// TwinCAT 3 PLC project stocker
// ProgramVersion: 3.1.4023.0
// CompilerDefines: VISU_USEWSTRING
// libraries:
//   CmpBitmapPool, * (System)
//   Tc2_MC2, * (Beckhoff Automation GmbH)
//   Tc2_Standard, * (Beckhoff Automation GmbH)
//   Tc2_System, * (Beckhoff Automation GmbH)
//   Tc2_Utilities, * (Beckhoff Automation GmbH)
//   Tc3_Module, * (Beckhoff Automation GmbH)
//   VisuDialogs, * (System)
//   VisuSymbols,3.5.10.0,System
// project tree:
//   DUTs/ENUM/ eP_alarmCode.TcDUT, eP_alarmLevel.TcDUT, eP_calculateMode.TcDUT, eP_direction.TcDUT, eP_ejevacMode.TcDUT, eP_eleMoveMode.TcDUT, eP_motionDirection.TcDUT, eP_programMode.TcDUT, eP_svMoveMode.TcDUT, eP_svType.TcDUT, eP_xyz.TcDUT
//   DUTs/REF/ ref_eje_input.TcDUT, ref_eje_io.TcDUT, ref_eje_output.TcDUT, ref_eje_param.TcDUT, ref_ele_input.TcDUT, ref_ele_io.TcDUT, ref_ele_output.TcDUT, ref_ele_param.TcDUT, ref_incjetInfo.TcDUT, ref_mc_moveAbs.TcDUT, ref_palletize.TcDUT, ref_productInfo.TcDUT, ref_sv_input.TcDUT, ref_sv_io.TcDUT, ref_sv_output.TcDUT, ref_sv_param.TcDUT, ref_teachingDetail.TcDUT, ref_teachPos.TcDUT, ref_cav.TcDUT, ref_upperLower.TcDUT, ref_XYZ.TcDUT
//   DUTs/ s_alarmList.TcDUT, s_DataSample.TcDUT, s_DataSampleCav.TcDUT, s_DataSampleCav_setQty.TcDUT, s_DataSampleGatelength.TcDUT, s_DataSamplePocketQty.TcDUT, s_gm_rotaryPos.TcDUT, s_DaraSampleSetQty.TcDUT, s_str_alarmList.TcDUT, s_timeSchedule.TcDUT, s_vels.TcDUT, s_velsXYZ.TcDUT
//   FBs/error/ fb_buzzerGenerater.TcPOU, fb_eventController.TcPOU, fb_eventListGenerator.TcPOU, fun_setAlarm.TcPOU
//   FBs/ fb_auto.TcPOU, fb_dataSampling.TcPOU, fb_debugData.TcPOU, fb_debuger.TcPOU, fb_gateLengthList.TcPOU, fb_getCav.TcPOU, fb_coordinateCal.TcPOU, fb_exchangeTraySystem.TcPOU, fb_IO.TcPOU, fb_jogController.TcPOU, fb_lsm_main.TcPOU, fb_manual.TcPOU, fb_mapping.TcPOU, fb_modeController.TcPOU, fb_motionController.TcPOU, fb_motorController.TcPOU, fb_oeprationChuck.TcPOU, fb_oeprationPush.TcPOU, fb_operationEjector.TcPOU, fb_operationElecylinder.TcPOU, fb_palletizeing.TcPOU, fb_paramInit.TcPOU, fb_productGenerator.TcPOU, fb_PTP.TcPOU, fb_recordingSystem.TcPOU, fb_sampleSchedule.TcPOU, fb_svControllers.TcPOU, fb_lensTranport.TcPOU, fb_text_control.TcPOU, fb_vacuumRetry.TcPOU, fb_eleControllers.TcPOU
//   FBs/fb_ejecter/ fb_ejector_io.TcPOU, fb_eje_controller.TcPOU, fb_eje_reset.TcPOU
//   FBs/fb_ele/ fb_ele_controller.TcPOU, fb_ele_io.TcPOU, fb_ele_reset.TcPOU
//   FBs/fb_sv/ fb_sv_controller.TcPOU, fb_sv_io.TcPOU, fb_sv_reset.TcPOU
//   FBs/gateMeasurementModule/ fb_gm_measurementModule.TcPOU, fb_gm_operationEjector.TcPOU, fb_gm_operationElecylinder.TcPOU, fb_gm_operationSV.TcPOU, fb_gm_PTP.TcPOU, fb_gm_removeLens.TcPOU, fb_gm_setting.TcPOU, fb_gm_transport.TcPOU
//   FBs/Incjet/ fb_incjetMapping.TcPOU
//   / GlobalTextList.TcGTLO, PlcTask.TcTTO, Visualization Manager.TcVMO (not stored), VISU_TASK.TcTTO
//   GVLs/ gvl_auto.TcGVL, gvl_axis.TcGVL, gvl_elecylinder.TcGVL, gvl_error.TcGVL, gvl_debug.TcGVL, gvl_gm.TcGVL, gvl_io.TcGVL, gvl_param.TcGVL, gvl_solv.TcGVL, gvl_text.TcGVL, gvl_visu.TcGVL
//   POUs/ MAIN.TcPOU
//   VISUs/Dialog/ d_gm_saveBtn.TcVIS, d_palletizeReset.TcVIS, d_preset.TcVIS, d_resetProject.TcVIS, d_sampleSchedule.TcVIS, d_saveBtn.TcVIS, d_saveProduct.TcVIS, d_saveSample.TcVIS, d_teahingDetail.TcVIS
//   VISUs/Sheet/ ImagePool.TcIPO (not stored), s_debug.TcVIS, s_gateLengthData.TcVIS, s_manual.TcVIS, s_addNewProduct.TcVIS, s_alarm.TcVIS, s_auto.TcVIS, s_gm_teaching.TcVIS, s_monitor.TcVIS, s_sample.TcVIS, s_setting.TcVIS, s_teaching1.TcVIS
// real-time tasks:
//   TASK PlcTask: cycle T#10ms, priority 20, ADS port 350
//   TASK VISU_TASK: cycle T#10ms, priority 30, ADS port 352
//   TASK VISU_TASK1: cycle T#10ms, priority 1, ADS port 351
// motion (NC):
//   TASK NC-Task 1 SAF: cycle T#2ms, priority 4, ADS port 501
//   TASK NC-Task 1 SVB: cycle T#10ms, priority 8, ADS port 511
//   AXIS lsm_axisX (id 1)
//     Velo: Maximum=5000
//     OtherSettings: AllowMotionCmdToSlave=true
//     encoder EncType=1
//       EncPara: ScaleFactorNumerator=54, ScaleFactorDenominator=10000, ReferenceSystem=1
//     drive DrvType=5
//       Analog: VeloReferenz=5200, TorqueSetpointScale=10, ScaleFactorActTorque=0.1
//       TimeComp: TaskDelayCycles=1
//     controller CtrType=1
//       CtrPara: PriorControlFactor=1
//         PosDiffControl: Enable=false
//         Observer: BandWidth=20
//   AXIS lsm_axisY (id 2)
//     Velo: Maximum=5000
//     OtherSettings: AllowMotionCmdToSlave=true
//     encoder EncType=1
//       EncPara: ScaleFactorNumerator=10, ScaleFactorDenominator=10000, ReferenceSystem=1
//     drive DrvType=5
//       Analog: VeloReferenz=5200, TorqueSetpointScale=10, ScaleFactorActTorque=0.1
//       TimeComp: TaskDelayCycles=1
//     controller CtrType=1
//       CtrPara: PriorControlFactor=1
//         PosDiffControl: Enable=false
//         Observer: BandWidth=20
//   AXIS lsm_axisZ (id 3)
//     Velo: Maximum=5000
//     OtherSettings: AllowMotionCmdToSlave=true
//     encoder EncType=1
//       EncPara: ScaleFactorNumerator=5, ScaleFactorDenominator=10000, ReferenceSystem=1
//     drive DrvType=5
//       Analog: VeloReferenz=5200, TorqueSetpointScale=10, ScaleFactorActTorque=0.1
//       TimeComp: TaskDelayCycles=1
//     controller CtrType=1
//       CtrPara: PriorControlFactor=1
//         PosDiffControl: Enable=false
//         Observer: BandWidth=20
//   AXIS gm_axisR (id 4)
//     General: UnitName=°
//     OtherSettings: AllowMotionCmdToSlave=true
//     encoder EncType=1
//       EncPara: ScaleFactorNumerator=20, ScaleFactorDenominator=10000, ReferenceSystem=1
//     drive DrvType=5
//       Analog: TorqueSetpointScale=10, ScaleFactorActTorque=0.1
//       TimeComp: TaskDelayCycles=1
//     controller CtrType=1
//       CtrPara: PriorControlFactor=1
//         Observer: BandWidth=20
// I/O:
//   DEVICE Device 1 (EtherCAT) (disabled), AmsNetId 192.168.8.53.2.1
//     Term 1 (EK1200) [EK1200-5000 EtherCAT Power supply (2A E-Bus)]
//       Term 2 (EL2088) [EL2088 8Ch. Dig. Output 24V, 0.5A, switching to negative]
//       Term 3 (EL1088) [EL1088 8Ch. Dig. Input 24V, 3ms, negative]
//       Term 4 (EK1110) [EK1110 EtherCAT extension]
//     Drive 5 (AZD4A-KED) [AZD4A-KED rev0301]
//     Box 6 (RCGW-ECT(32Byte/32Byte)) [RCGW-ECT(32Byte/32Byte)]
//     Box 7 (CU1128) [CU1128 6x EtherCAT junction]
//       Term 8 (EK1100) [EK1100 EtherCAT Coupler (2A E-Bus)]
//         Term 9 (EL2889) [EL2889 16Ch. Dig. Output 24V, 0.5A, negative]
//         Term 10 (EL2088) [EL2088 8Ch. Dig. Output 24V, 0.5A, switching to negative]
//         Term 11 (EL1889) [EL1889 16Ch. Dig. Input 24V, 3ms, negative]
//         Term 12 (EL1088) [EL1088 8Ch. Dig. Input 24V, 3ms, negative]
//         Term 17 (EL9011) [EL9011 End Terminal]
//       Box 13 (DL-EC1A) [DL-EC1A]
//       Box 14 (ECCBP88N) [ECCBP Digital 8 Inputs/8 Outputs Unit (NPN)]
//       Term 15 (CU1128-B) [CU1128 6x EtherCAT junction - Dev A]
//       Term 16 (CU1128-C) [CU1128 6x EtherCAT junction - Dev B]
// variable links:
//   stocker/stocker Instance <-> Device 1 (EtherCAT)/Box 6 (RCGW-ECT(32Byte/32Byte))
//     PlcTask Inputs/gvl_io.in_wire_ele_gateMeasurement <-> In/IN02
//     PlcTask Inputs/gvl_io.in_wire_ele_stocker <-> In/IN01
//     PlcTask Outputs/gvl_io.out_wire_ele_gateMeasurement <-> Out/OUT02
//     PlcTask Outputs/gvl_io.out_wire_ele_stocker <-> Out/OUT01
//   stocker/stocker Instance <-> Device 1 (EtherCAT)/Box 7 (CU1128)/Box 13 (DL-EC1A)
//     PlcTask Inputs/gvl_io.in_wire_gateLength <-> ID01 Current Value/ID01 Current Value (P.V.)
//     PlcTask Inputs/gvl_io.in_wire_gateMeasurementStatus <-> Status of System/Error Status
//   stocker/stocker Instance <-> Device 1 (EtherCAT)/Box 7 (CU1128)/Box 14 (ECCBP88N)
//     PlcTask Inputs/gvl_io.in_bitNumber{0..3} <-> TxPDO1/DI{4..7}  (4 links)
//     PlcTask Inputs/gvl_io.in_wire_dummySignal <-> TxPDO1/DI2
//     PlcTask Inputs/gvl_io.in_wire_gatelengthIsSuccessed <-> TxPDO1/DI1
//     PlcTask Inputs/gvl_io.in_wire_lensSetDone <-> TxPDO1/DI0
//     PlcTask Outputs/gvl_io.out_wire_requestLens <-> RxPDO1/DO0
//   stocker/stocker Instance <-> Device 1 (EtherCAT)/Box 7 (CU1128)/Term 8 (EK1100)/Term 10 (EL2088)
//     PlcTask Outputs/gvl_io.out_wire_gm_svPickUp <-> Channel 3/Output
//     PlcTask Outputs/gvl_io.out_wire_gm_svRotary <-> Channel 5/Output
//     PlcTask Outputs/gvl_io.out_wire_gm_svStamp <-> Channel 1/Output
//   stocker/stocker Instance <-> Device 1 (EtherCAT)/Box 7 (CU1128)/Term 8 (EK1100)/Term 11 (EL1889)
//     PlcTask Inputs/gvl_io.in_wire_ejectorBrk <-> Channel 9/Input
//     PlcTask Inputs/gvl_io.in_wire_ejectorVac <-> Channel 8/Input
//     PlcTask Inputs/gvl_io.in_wire_fiberSens <-> Channel 14/Input
//     PlcTask Inputs/gvl_io.in_wire_gm_ejectorBrk <-> Channel 2/Input
//     PlcTask Inputs/gvl_io.in_wire_gm_ejectorVac <-> Channel 1/Input
//     PlcTask Inputs/gvl_io.in_wire_gm_fiberSens <-> Channel 7/Input
//     PlcTask Inputs/gvl_io.in_wire_gm_svChuckClose <-> Channel 6/Input
//     PlcTask Inputs/gvl_io.in_wire_gm_svChuckOpen <-> Channel 5/Input
//     PlcTask Inputs/gvl_io.in_wire_gm_svPushClose <-> Channel 4/Input
//     PlcTask Inputs/gvl_io.in_wire_gm_svPushOpen <-> Channel 3/Input
//     PlcTask Inputs/gvl_io.in_wire_incjet_error <-> Channel 16/Input
//     PlcTask Inputs/gvl_io.in_wire_incjet_ready <-> Channel 15/Input
//     PlcTask Inputs/gvl_io.in_wire_svChuckClose <-> Channel 11/Input
//     PlcTask Inputs/gvl_io.in_wire_svChuckOpen <-> Channel 10/Input
//     PlcTask Inputs/gvl_io.in_wire_svPushClose <-> Channel 13/Input
//     PlcTask Inputs/gvl_io.in_wire_svPushOpen <-> Channel 12/Input
//   stocker/stocker Instance <-> Device 1 (EtherCAT)/Box 7 (CU1128)/Term 8 (EK1100)/Term 12 (EL1088)
//     PlcTask Inputs/gvl_io.in_wire_gm_svPickUpMoving <-> Channel 4/Input
//     PlcTask Inputs/gvl_io.in_wire_gm_svPickUpOrigin <-> Channel 3/Input
//     PlcTask Inputs/gvl_io.in_wire_gm_svRotaryMoving <-> Channel 6/Input
//     PlcTask Inputs/gvl_io.in_wire_gm_svRotaryOrigin <-> Channel 5/Input
//     PlcTask Inputs/gvl_io.in_wire_gm_svStampMoving <-> Channel 2/Input
//     PlcTask Inputs/gvl_io.in_wire_gm_svStampOrigin <-> Channel 1/Input
//   stocker/stocker Instance <-> Device 1 (EtherCAT)/Box 7 (CU1128)/Term 8 (EK1100)/Term 9 (EL2889)
//     PlcTask Outputs/gvl_io.out_wire_ejectorBrk <-> Channel 9/Output
//     PlcTask Outputs/gvl_io.out_wire_ejectorVac <-> Channel 8/Output
//     PlcTask Outputs/gvl_io.out_wire_gm_ejectorBrk <-> Channel 2/Output
//     PlcTask Outputs/gvl_io.out_wire_gm_ejectorVac <-> Channel 1/Output
//     PlcTask Outputs/gvl_io.out_wire_gm_svCPush <-> Channel 3/Output
//     PlcTask Outputs/gvl_io.out_wire_gm_svChuck <-> Channel 5/Output
//     PlcTask Outputs/gvl_io.out_wire_incjet_stampDeny <-> Channel 16/Output
//     PlcTask Outputs/gvl_io.out_wire_svCPush <-> Channel 12/Output
//     PlcTask Outputs/gvl_io.out_wire_svChuck <-> Channel 10/Output
//   stocker/stocker Instance <-> Device 1 (EtherCAT)/Term 1 (EK1200)/Term 2 (EL2088)
//     PlcTask Outputs/gvl_io.out_wire_saftyUnitReset <-> Channel 1/Output
//     PlcTask Outputs/gvl_io.out_wire_signalTowerBuzzer <-> Channel 5/Output
//     PlcTask Outputs/gvl_io.out_wire_signalTowerGreen <-> Channel 4/Output
//     PlcTask Outputs/gvl_io.out_wire_signalTowerRed <-> Channel 2/Output
//     PlcTask Outputs/gvl_io.out_wire_signalTowerYellow <-> Channel 3/Output
//   stocker/stocker Instance <-> Device 1 (EtherCAT)/Term 1 (EK1200)/Term 3 (EL1088)
//     PlcTask Inputs/gvl_io.in_wire_frontSaftyDoor <-> Channel 3/Input
//     PlcTask Inputs/gvl_io.in_wire_saftyUnitState <-> Channel 1/Input
//   stocker/stocker Instance <-> NC-Task 1 SAF/Axes/gm_axisR
//     PlcTask Inputs/gvl_axis.axisR.NcToPlc <-> Outputs/ToPlc
//     PlcTask Outputs/gvl_axis.axisR.PlcToNc <-> Inputs/FromPlc
//   stocker/stocker Instance <-> NC-Task 1 SAF/Axes/lsm_axisX
//     PlcTask Inputs/gvl_axis.axisX.NcToPlc <-> Outputs/ToPlc
//     PlcTask Outputs/gvl_axis.axisX.PlcToNc <-> Inputs/FromPlc
//   stocker/stocker Instance <-> NC-Task 1 SAF/Axes/lsm_axisY
//     PlcTask Inputs/gvl_axis.axisY.NcToPlc <-> Outputs/ToPlc
//     PlcTask Outputs/gvl_axis.axisY.PlcToNc <-> Inputs/FromPlc
//   stocker/stocker Instance <-> NC-Task 1 SAF/Axes/lsm_axisZ
//     PlcTask Inputs/gvl_axis.axisZ.NcToPlc <-> Outputs/ToPlc
//     PlcTask Outputs/gvl_axis.axisZ.PlcToNc <-> Inputs/FromPlc

CONFIGURATION stocker
    RESOURCE PLC ON TwinCAT3
        TASK PlcTask(INTERVAL := T#10ms, PRIORITY := 20);
        TASK VISU_TASK(INTERVAL := T#10ms, PRIORITY := 40);
        PROGRAM MAIN WITH PlcTask : MAIN;
        PROGRAM VisuElems_Visu_Prg WITH VISU_TASK : VisuElems.Visu_Prg;
    END_RESOURCE
END_CONFIGURATION

// ---- DUTs/ENUM/eP_alarmCode.TcDUT
{attribute 'qualified_only'}
{attribute 'strict'}
TYPE eP_alarmCode :
(
	_ := 0,
	A,
	E,
	M,
	GM,
	W
);
END_TYPE

// ---- DUTs/ENUM/eP_alarmLevel.TcDUT
{attribute 'qualified_only'}
{attribute 'strict'}
TYPE eP_alarmLevel :
(
	NONE := 0,
	INFO := 1,
	WARNING := 2,
	ERROR := 3
);
END_TYPE

// ---- DUTs/ENUM/eP_calculateMode.TcDUT
{attribute 'qualified_only'}
{attribute 'strict'}
TYPE eP_calculateMode :
(
	Affine := 0,
	Homography := 1
);
END_TYPE

// ---- DUTs/ENUM/eP_direction.TcDUT
{attribute 'qualified_only'}
{attribute 'strict'}
TYPE eP_direction :
(
	keep :=0,
	negative,
	positive
);
END_TYPE

// ---- DUTs/ENUM/eP_ejevacMode.TcDUT
{attribute 'qualified_only'}
{attribute 'strict'}
TYPE eP_ejevacMode :
(
	vacON := 1,
	vacOff := 2,
	break := 3,
	breakOff := 4,
	halt := 0
);
END_TYPE

// ---- DUTs/ENUM/eP_eleMoveMode.TcDUT
{attribute 'qualified_only'}
{attribute 'strict'}
TYPE eP_eleMoveMode :
(
	eleA := 1,
	eleB :=-1,
	stop := 0
);
END_TYPE

// ---- DUTs/ENUM/eP_motionDirection.TcDUT
{attribute 'qualified_only'}
{attribute 'strict'}
TYPE eP_motionDirection :
(
	XYZ := 1,
	ZYX := -1,
	Y_X_Z := 2,
	Z_X_Y := -2
);
END_TYPE

// ---- DUTs/ENUM/eP_programMode.TcDUT
{attribute 'qualified_only'}
{attribute 'strict'}
TYPE eP_programMode :
(
	manual := 0,
	auto,
	error
);
END_TYPE

// ---- DUTs/ENUM/eP_svMoveMode.TcDUT
{attribute 'qualified_only'}
{attribute 'strict'}
TYPE eP_svMoveMode :
(
	svA := 1,
	svB := -1,
	stop := 0
);
END_TYPE

// ---- DUTs/ENUM/eP_svType.TcDUT
{attribute 'qualified_only'}
{attribute 'strict'}
TYPE eP_svType :
(
	single,
	double
);
END_TYPE

// ---- DUTs/ENUM/eP_xyz.TcDUT
{attribute 'qualified_only'}
{attribute 'strict'}
TYPE eP_xyz :
(
	x := 0,
	y,
	z
);
END_TYPE

// ---- DUTs/REF/ref_eje_input.TcDUT
TYPE ref_eje_input :
STRUCT
	in_flg_sensVac : BOOL;
	in_flg_sensBrk : BOOL;
END_STRUCT
END_TYPE

// ---- DUTs/REF/ref_eje_io.TcDUT
TYPE ref_eje_io :
STRUCT
	param:	ref_eje_param;
	input:	ref_eje_input;
	output:	ref_eje_output;
END_STRUCT
END_TYPE

// ---- DUTs/REF/ref_eje_output.TcDUT
TYPE ref_eje_output :
STRUCT
	out_flg_ejeVac : BOOL;
	out_flg_ejeBrk : BOOL;
END_STRUCT
END_TYPE

// ---- DUTs/REF/ref_eje_param.TcDUT
TYPE ref_eje_param :
STRUCT
	var_mutex : INT;
	var_timeOut : TIME;
	var_BrkTime : TIME;
	flg_reset :BOOL;
END_STRUCT
END_TYPE

// ---- DUTs/REF/ref_ele_input.TcDUT
TYPE ref_ele_input :
STRUCT
	in_flg_sensA : BOOL;
	in_flg_sensB : BOOL;
	in_flg_sensNone : BOOL;
	in_wire_error : bool;
END_STRUCT
END_TYPE

// ---- DUTs/REF/ref_ele_io.TcDUT
TYPE ref_ele_io :
STRUCT
	param:	ref_ele_param;
	input:	ref_ele_input;
	output:	ref_ele_output;
END_STRUCT
END_TYPE

// ---- DUTs/REF/ref_ele_output.TcDUT
TYPE ref_ele_output :
STRUCT
	out_flg_eleA : BOOL;
	out_flg_eleB : BOOL;
	out_flg_reset : BOOL;
END_STRUCT
END_TYPE

// ---- DUTs/REF/ref_ele_param.TcDUT
TYPE ref_ele_param :
STRUCT
	var_mutex : INT;
	var_timeOut : TIME;
	flg_reset :BOOL;
END_STRUCT
END_TYPE

// ---- DUTs/REF/ref_incjetInfo.TcDUT
TYPE ref_incjetInfo :
STRUCT
	var_msgNo : INT;
	flg_denyStamp : BOOL;
	flg_numberingReset : BOOL;
	flg_numberingCount : BOOL;
	flg_numberingStop : BOOL;
	flg_warningReset : BOOL;
	flg_stampReady : BOOL;
	flg_incLow : BOOL;
	flg_incOut : BOOL;
	flg_error : BOOL;
	flg_busy : BOOL;
	flg_stampRun : BOOL;
	flg_heatUpDone : BOOL;
	flg_systemRun : BOOL;
	flg_stampsDone : BOOL;
	flg_numberingCountDone : BOOL;
	flg_fluxLow : BOOL;
	flg_incFluxLow : BOOL;
	flg_headCoverIsOpen : BOOL;
	flg_stampDone : BOOL;
END_STRUCT
END_TYPE

// ---- DUTs/REF/ref_mc_moveAbs.TcDUT
TYPE ref_mc_moveAbs :
STRUCT
	Execute      : BOOL;
    Position     : LREAL; 
    Velocity     : LREAL; 
    Acceleration : LREAL; 
    Deceleration : LREAL; 
    Jerk         : LREAL;
    BufferMode   : MC_BufferMode;
    Options      : ST_MoveOptions;
	Done           : BOOL;
    Busy           : BOOL;
    Active         : BOOL;
    CommandAborted : BOOL;
    Error          : BOOL;
    ErrorID        : UDINT;
END_STRUCT
END_TYPE

// ---- DUTs/REF/ref_palletize.TcDUT
TYPE ref_palletize :
STRUCT
	Pos : ARRAY[1..4] OF ref_xyz ;
	teachingDetail : ref_teachingDetail;
	teachingDetailVels : s_velsXYZ;
END_STRUCT
END_TYPE

// ---- DUTs/REF/ref_productInfo.TcDUT
TYPE ref_productInfo :
STRUCT
	num : INT;
	name : STRING;
	cavQty : INT;
	bottomPocketQty : INT;
	vertivalPocketQty : INT ;
	pocketSumQty : INT;
	startCav : INT;
	gateLength_min : INT;
	gateLength_max : INT;
	teachPos : ref_teachPos;
	autoVels : s_velsXYZ;
	manaulVels : s_velsXYZ;
	incjetMsgNo : INT;
	flg_mode_stocker: BOOL;
	flg_mode_measurement: BOOL;
END_STRUCT
END_TYPE

// ---- DUTs/REF/ref_sv_input.TcDUT
TYPE ref_sv_input :
STRUCT
	in_flg_sensA:	BOOL;
	in_flg_sensB:	BOOL;
END_STRUCT
END_TYPE

// ---- DUTs/REF/ref_sv_io.TcDUT
TYPE ref_sv_io :
STRUCT
	param: ref_sv_param;
	in: ref_sv_input;
	out:ref_sv_output;
END_STRUCT
END_TYPE

// ---- DUTs/REF/ref_sv_output.TcDUT
TYPE ref_sv_output :
STRUCT
	out_flg_svA:	BOOL;
	out_flg_svB:	BOOL;
END_STRUCT
END_TYPE

// ---- DUTs/REF/ref_sv_param.TcDUT
TYPE ref_sv_param :
STRUCT
	var_svType:ep_svType;
	var_mutex : INT;
	var_timeOut : TIME;
	flg_reset :BOOL;
END_STRUCT
END_TYPE

// ---- DUTs/REF/ref_teachingDetail.TcDUT
TYPE ref_teachingDetail :
STRUCT
	passingPos : ref_XYZ;
	settingPos : ref_XYZ;
END_STRUCT
END_TYPE

// ---- DUTs/REF/ref_teachPos.TcDUT
TYPE ref_teachPos :
STRUCT
	palletize : ref_upperLower;
	initial : ref_xyz;
	pickUp : ref_xyz;
	remove :ref_xyz;
	sample  : ARRAY[1..8] OF ref_xyz;
	gm_rotary	: s_gm_rotaryPos;
END_STRUCT
END_TYPE

// ---- DUTs/REF/ref_cav.TcDUT
TYPE ref_cav :
STRUCT
	cav : ARRAY [1..8] OF  ref_palletize;
END_STRUCT
END_TYPE

// ---- DUTs/REF/ref_upperLower.TcDUT
TYPE ref_upperLower :
STRUCT
	upperLower : ARRAY[1..2] OF ref_cav ;
END_STRUCT
END_TYPE

// ---- DUTs/REF/ref_XYZ.TcDUT
TYPE ref_XYZ :
STRUCT
	x : LREAL ;
	y : LREAL ;
	z : LREAL ;
END_STRUCT
END_TYPE

// ---- DUTs/s_alarmList.TcDUT
TYPE s_alarmList :
STRUCT
	var_alarmLevel : eP_alarmLevel;
	var_alarmName : WSTRING;
	var_alarmMassge : WSTRING;
	var_alarmTime : DT;
	var_alarmCode1 : eP_alarmCode;
	var_alarmCode2 : UDINT;
	
END_STRUCT
END_TYPE

// ---- DUTs/s_DataSample.TcDUT
TYPE s_DataSample :
STRUCT
	DataSet :  ARRAY[0..500] OF s_DataSampleCav;
	SetQty	:  s_DataSampleCav_setQty;
END_STRUCT
END_TYPE

// ---- DUTs/s_DataSampleCav.TcDUT
TYPE s_DataSampleCav :
STRUCT
	cav : ARRAY[0..8] OF s_DataSamplePocketQty;
END_STRUCT
END_TYPE

// ---- DUTs/s_DataSampleCav_setQty.TcDUT
TYPE s_DataSampleCav_setQty :
STRUCT
	cav : ARRAY[0..8] OF  s_DaraSampleSetQty;
END_STRUCT
END_TYPE

// ---- DUTs/s_DataSampleGatelength.TcDUT
TYPE s_DataSampleGatelength :
STRUCT
	gateLength	: LREAL;
	setDate		: STRING;
END_STRUCT
END_TYPE

// ---- DUTs/s_DataSamplePocketQty.TcDUT
TYPE s_DataSamplePocketQty :
STRUCT
	pocketNo : ARRAY[0..100] OF s_DataSampleGatelength;
END_STRUCT
END_TYPE

// ---- DUTs/s_gm_rotaryPos.TcDUT
TYPE s_gm_rotaryPos :
STRUCT
	origin	: LREAL;
	pickUp	: LREAL;
	set		: LREAL;
	remove  : LREAL;
END_STRUCT
END_TYPE

// ---- DUTs/s_DaraSampleSetQty.TcDUT
TYPE s_DaraSampleSetQty :
STRUCT
	nonDefectiveQty : INT;
	defectiveQty	:INT;
END_STRUCT
END_TYPE

// ---- DUTs/s_str_alarmList.TcDUT
TYPE s_str_alarmList :
STRUCT
	var_alarmLevel : STRING;
	var_alarmName : WSTRING;
	var_alarmMassge : WSTRING;
	var_alarmTime : STRING;
	var_alarmCode1 : eP_alarmCode;
	var_alarmCode2 : STRING;
	
END_STRUCT
END_TYPE

// ---- DUTs/s_timeSchedule.TcDUT
TYPE s_timeSchedule :
STRUCT
	hour : WORD;
	minute: WORD;
END_STRUCT
END_TYPE

// ---- DUTs/s_vels.TcDUT
TYPE s_vels :
STRUCT
	vel : LREAL := 20;
	acc : LREAL := 20;
	dcc : LREAL := 20;
END_STRUCT
END_TYPE

// ---- DUTs/s_velsXYZ.TcDUT
TYPE s_velsXYZ :
STRUCT
	x : s_vels;
	y : s_vels;
	z : s_vels;
END_STRUCT
END_TYPE

// ---- GVLs/gvl_auto.TcGVL
{attribute 'qualified_only'}
VAR_GLOBAL
	gateLengthIsPassed		: BOOL;
	requirementToPickUpLens	: BOOL;
	pickUpLnesDone			: BOOL;
	chuckopenDone			: BOOL;
	lensVacuumDone			: BOOL;
	cavNo					: INT;
	buf_cavNo				: INT ;
	autoModeStop			: BOOL;
	autoModeStoped			: BOOL;
	motorPowerOn			: BOOL;
	flg_trayChangeDone		: BOOL;
	gm_rotaryPowerOn		: BOOL;
	flg_gateData_Tx			: BOOL;
	flg_gm_measurementClosed: BOOL;
	flg_gm_transportClosed	: BOOL;
	flg_transportClosed		: BOOL;
	flg_VacuumRetry			: BOOL;
	flg_gm_VacuumRetry		: BOOL;
	flg_DataSample_nonDefective: BOOL;
	flg_DataSample_defective: BOOL;
	flg_DataSamle_sample: BOOL;
	buf_gateLength: LREAL;
	flg_dataSampling_run: BOOL;
	var_DataSet				: s_DataSample; //lateset data is var_DataSet[0], oldest is var_DataSet[500], cav[0] and pocketNo[0] are unused
	flg_gm_eleIsDown: BOOL;
	flg_axisIsPcikingUp: BOOL;
	flg_buf_gateLengthIsPassed: BOOL;
	flg_gateLength: BOOL;
	flg_sampling: BOOL;
END_VAR
VAR_GLOBAL PERSISTENT
	pocketNo				: ARRAY[0..8] OF INT;
	var_defectiveLens		: ARRAY[0..8] OF INT;
	
	flg_pocketCountCheck_cav: int;
	flg_pocketCountCheck: BOOL;
END_VAR

// ---- GVLs/gvl_axis.TcGVL
{attribute 'qualified_only'}
VAR_GLOBAL
	axisX : AXIS_REF;
	axisY : AXIS_REF;
	axisZ : AXIS_REF;
	axisR : AXIS_REF;
	
	fbi_mc_powerX :MC_Power;
	fbi_mc_powerY :MC_Power;
	fbi_mc_powerZ :MC_Power;
	fbi_mc_powerR :MC_Power;
	
	fbi_mc_absX : MC_MoveAbsolute;
	fbi_mc_absY : MC_MoveAbsolute;
	fbi_mc_absZ : MC_MoveAbsolute;
	fbi_mc_absR : MC_MoveAbsolute;
	
	ref_x : ref_mc_moveAbs;
	ref_y : ref_mc_moveAbs;
	ref_z : ref_mc_moveAbs;
	ref_r : ref_mc_moveAbs;
	
	fbi_mc_jogX : MC_Jog;
	fbi_mc_jogY : MC_Jog;
	fbi_mc_jogZ : MC_Jog;
	fbi_mc_jogR : MC_Jog;
	
	fbi_motionControler: fb_motionController;
	
	flg_motorReady: BOOL;
END_VAR

// ---- GVLs/gvl_elecylinder.TcGVL
{attribute 'qualified_only'}
VAR_GLOBAL
	
	fbi_axisTransport 		: fb_ele_controller;
	fbi_axisSample 			: fb_ele_controller;
	fbi_axisTrayChange 		: fb_ele_controller;
	fbi_axisRotary 			: fb_ele_controller;
	fbi_gm_axisTransport 	: fb_ele_controller;
	fbi_gm_axisPickUp 		: fb_ele_controller;
	

	ref_axis_transport 		: ref_ele_io;
	ref_axis_sample		 	: ref_ele_io;
	ref_axis_trayChange 	: ref_ele_io;
	ref_axis_rotary 		: ref_ele_io;
	ref_gm_axisTransport 	: ref_ele_io;
	ref_gm_axisPickUp 		: ref_ele_io;
END_VAR

// ---- GVLs/gvl_error.TcGVL
{attribute 'qualified_only'}
VAR_GLOBAL
	var_ary_alarmlistActive 	: ARRAY[1..10] OF s_str_alarmList;
	flg_error					: BOOL;
	flg_warning					: BOOL;
	flg_info					: BOOL;
	flg_reset					: BOOL;
	flg_alramBusy				: BOOL;
	
	flg_fiberSens 				: BOOL;
	flg_vacuum					: BOOL;
	flg_axisXTorqueOver			: BOOL;
	flg_axisYTorqueOver			: BOOL;
	flg_axisZTorqueOver			: BOOL;
	flg_axisRTorqueOver			: BOOL;
	
	flg_resetEventFlg			: BOOL;
	flg_eventDisplayRest		: BOOL;
	flg_ararmLevelRest			: BOOL;
	flg_gm_fiberSens			: BOOL;
	flg_trayChangeError			: BOOL;
	flg_incjet					: BOOL;
	
	flg_sample_windown_warning  : BOOL;
	flg_sample_windown_error	: BOOL;
END_VAR
VAR_GLOBAL PERSISTENT
	var_ary_alarmlistLog 		: ARRAY[1..50] OF s_alarmList;
END_VAR

// ---- GVLs/gvl_debug.TcGVL
{attribute 'qualified_only'}
VAR_GLOBAL
	gateLengthISSuccessed	: BOOL;
	dummySignal				: BOOL;
	lensSetDone				: BOOL;
	flg_debug_run			: BOOL;
	var_cav					: INT;
	out_busy			    : BOOL;
	out_lensSetDone			: BOOL;
	out_fiberSens			: BOOL;
	cavConecctSkip			: BOOL;
	flg_passingMeasurement	: BOOL;
	flg_stampReady: BOOL;
	flg_stampDone: BOOL;
	flg_check_quality: BOOL;
	flg_to_measurement : BOOL;
	flg_to_stocker : BOOL;
	flg_to_demand: BOOL;
	flg_to_acquired: BOOL;
	
END_VAR

// ---- GVLs/gvl_gm.TcGVL
{attribute 'qualified_only'}
VAR_GLOBAL
	
	flg_lensSetDoneFromGM		: BOOL;
	flg_lensPickUpDone			: BOOL;
	flg_requestPickup			: BOOL;
	flg_lensRequest				: BOOL;
	
	var_buf_measurementCav		: INT;
	var_buf_tranportCav			: INT;
	flg_gateLengthIsPassed: BOOL;
	flg_buf_gateLengthIsPassed: BOOL;
END_VAR
VAR_GLOBAL PERSISTENT
	var_buf_manualVel			: LREAL;
	var_buf_autoVel				: LREAL;
	var_buf_autoAcc				: LREAL;
	var_buf_autoDec				: LREAL;
	var_rotaryPos 				: s_gm_rotaryPos;
	var_incjetInfo				:ref_incjetInfo;
END_VAR

// ---- GVLs/gvl_io.TcGVL
{attribute 'qualified_only'}
VAR_GLOBAL
	in_wire_saftyCircuitState				AT %I* : BOOL;
	in_wire_saftyUnitState					AT %I* : BOOL;
	in_wire_frontSaftyDoor					AT %I* : BOOL;
	in_wire_btnGreen						AT %I* : BOOL;
	in_wire_btnRed							AT %I* : BOOL;
	in_bitNumber0							AT %I* : BOOL;
	in_bitNumber1							AT %I* : BOOL;
	in_bitNumber2							AT %I* : BOOL;
	in_bitNumber3							AT %I* : BOOL;
	in_wire_gateLengthIsFailed				AT %I* : BOOL;
	in_wire_lensSetDone						AT %I* : BOOL;
	in_wire_gatelengthIsSuccessed			AT %I* : BOOL;
	in_wire_dummySignal						AT %I* : BOOL;
	in_wire_fiberSens						AT %I* : BOOL;
	in_wire_gm_fiberSens					AT %I* : BOOL;
	//solv
	in_wire_ejectorVac						AT %I* : BOOL;
	in_wire_ejectorBrk						AT %I* : BOOL;
	in_wire_svChuckClose					AT %I* : BOOL;
	in_wire_svChuckOpen						AT %I* : BOOL;
	in_wire_svPushClose						AT %I* : BOOL;
	in_wire_svPushOpen						AT %I* : BOOL;
	in_wire_gm_ejectorVac					AT %I* : BOOL;
	in_wire_gm_ejectorBrk					AT %I* : BOOL;
	in_wire_gm_svChuckClose					AT %I* : BOOL;
	in_wire_gm_svChuckOpen					AT %I* : BOOL;
	in_wire_gm_svPushClose					AT %I* : BOOL;
	in_wire_gm_svPushOpen					AT %I* : BOOL;
	in_wire_gm_svRotaryOrigin				AT %I* : BOOL;
	in_wire_gm_svRotaryMoving				AT %I* : BOOL;
	in_wire_gm_svPickUpOrigin				AT %I* : BOOL;
	in_wire_gm_svPickUpMoving				AT %I* : BOOL;
	in_wire_gm_svStampOrigin				AT %I* : BOOL;
	in_wire_gm_svStampMoving				AT %I* : BOOL;
	//elecylinder
	in_wire_ele_stocker						AT %I* : UINT;
	in_wire_ele_gateMeasurement				AT %I* : UINT;
	
	in_wire_incjet_ready					AT %I* : BOOL;
	in_wire_incjet_run  					AT %I* : BOOL;
	in_wire_incjet_error					AT %I* : BOOL;
	
	in_flg_eleTransportOrigin						: BOOL;
	in_flg_eleTransportMoving						: BOOL;
	in_flg_eleTransportError						: BOOL;
	in_flg_eleSampleOrigin							: BOOL;
	in_flg_eleSampleMoving							: BOOL;
	in_flg_eleSampleError							: BOOL;
	in_flg_eleTrayChangeOrigin						: BOOL;
	in_flg_eleTrayChangeMoving						: BOOL;
	in_flg_eleTrayChangeError						: BOOL;
	in_flg_eleRotaryOrigin							: BOOL;
	in_flg_eleRotaryMoving							: BOOL;
	in_flg_eleRotaryError							: BOOL;
	in_flg_gm_elePickupOrigin						: BOOL;
	in_flg_gm_elePickupMoving						: BOOL;
	in_flg_gm_elePickupError						: BOOL;
	in_flg_gm_eleTransportOrigin					: BOOL;
	in_flg_gm_eleTransportMoving					: BOOL;
	in_flg_gm_eleTransPortError						: BOOL;
	
	
	
	in_wire_gateLength						AT %I* : DINT;
	in_wire_gateMeasurementStatus			AT %I* : BOOL;
	in_wire_gateMeasurementErrCode			AT %I* : UINT;
	out_wire_gateMeasurementReset			AT %Q* : DINT;
	out_wire_gateMeasurementPreset			AT %Q* : DINT;
	
	out_wire_saftyUnitReset					AT %Q* : BOOL;
	out_wire_signalTowerRed 				AT %Q* : BOOL;
	out_wire_signalTowerGreen 				AT %Q* : BOOL;
	out_wire_signalTowerYellow				AT %Q* : BOOL;
	out_wire_signalTowerBuzzer 				AT %Q* : BOOL;
	
	out_wire_requestLens					AT %Q* : BOOL;
	//solv
	out_wire_ejectorVac						AT %Q* : BOOL;
	out_wire_ejectorBrk						AT %Q* : BOOL;
	out_wire_svChuck						AT %Q* : BOOL;
	out_wire_svCPush						AT %Q* : BOOL;
	out_wire_gm_ejectorVac					AT %Q* : BOOL;
	out_wire_gm_ejectorBrk					AT %Q* : BOOL;
	out_wire_gm_svChuck						AT %Q* : BOOL;
	out_wire_gm_svCPush						AT %Q* : BOOL;
	out_wire_gm_svRotary					AT %Q* : BOOL;
	out_wire_gm_svPickUp					AT %Q* : BOOL;
	out_wire_gm_svStamp						AT %Q* : BOOL;

	//elecylinder
	out_wire_ele_stocker					AT %Q* : UINT;
	out_wire_ele_gateMeasurement			AT %Q* : UINT;
	
	out_wire_incjet_stampDeny				AT %Q* : BOOL;
	
	out_flg_eleTransportOrigin						: BOOL;
	out_flg_eleTransportMoving						: BOOL;
	out_flg_eleTransportReset						: BOOL;
	out_flg_eleSampleOrigin							: BOOL;
	out_flg_eleSampleMoving							: BOOL;
	out_flg_eleSampleReset							: BOOL;
	out_flg_eleTrayChangeOrigin						: BOOL;
	out_flg_eleTrayChangeMoving						: BOOL;
	out_flg_eleTrayChangeReset						: BOOL;
	out_flg_eleRotaryOrigin							: BOOL;
	out_flg_eleRotaryMoving							: BOOL;
	out_flg_eleRotaryReset							: BOOL;
	out_flg_gm_elePickupOrigin						: BOOL;
	out_flg_gm_elePickupMoving						: BOOL;
	out_flg_gm_elePickupReset						: BOOL;
	out_flg_gm_eleTransportOrigin					: BOOL;
	out_flg_gm_eleTransportMoving					: BOOL;
	out_flg_gm_eleTransPortReset					: BOOL;
	flg_bitNumber0									: BOOL;
	flg_bitNumber1									: BOOL;
	flg_bitNumber2									: BOOL;
	flg_bitNumber3									: BOOL;
	flg_dummySiganl									: BOOL;
	flg_gateLengthIsSuccessed						: BOOL;
	flg_lensSetDone									: BOOL;
	flg_fiberSens									: BOOL;
	flg_btnGreen									: BOOL;
	flg_btnRed										: BOOL;
	flg_frontSaftyDoor								: BOOL;
	var_gateLength									: DINT;
	flg_gatemeasurementStatus						: BOOL;
	var_gateMeasurementErrCode						: UDINT;
	var_gateMeasurementReset						: DINT;
	var_gateMeasurementPreset						: DINT;
	flg_gm_fiberSens								: BOOL;
	flg_saftyUnitState								: BOOL;
	flg_saftyUnitReset								: BOOL;
	flg_requestLens									: BOOL;
	flg_signalTowerBuzzer							: BOOL;
	flg_signalTowerGreen							: BOOL;
	flg_signalTowerRed								: BOOL;
	flg_signalTowerYellow							: BOOL;

END_VAR

// ---- GVLs/gvl_param.TcGVL
{attribute 'qualified_only'}
VAR_GLOBAL
	var_currentMode 		: eP_programMode;
	var_currentTrayPos 		: INT;
END_VAR
VAR_GLOBAL PERSISTENT
	var_productInfo 		: ARRAY [0..10] OF ref_productInfo;
	var_currentProductID 	: INT := 0;
	var_b					: INT;
END_VAR

// ---- GVLs/gvl_solv.TcGVL
{attribute 'qualified_only'}
VAR_GLOBAL	
	fbi_ejector 	: fb_eje_controller;
	fbi_chuck 		: fb_sv_controller;
	fbi_push 		: fb_sv_controller;
	fbi_gm_ejector 	: fb_eje_controller;
	fbi_gm_chuck 	: fb_sv_controller;
	fbi_gm_push 	: fb_sv_controller;
	fbi_gm_rotary 	: fb_sv_controller;
	fbi_gm_pickup 	: fb_sv_controller;
	fbi_gm_stamp 	: fb_sv_controller;

	ref_ejector 	: ref_eje_io;
	ref_chuck 		: ref_sv_io;
	ref_push 		: ref_sv_io;
	ref_gm_ejctor 	: ref_eje_io;
	ref_gm_chuck 	: ref_sv_io;
	ref_gm_push 	: ref_sv_io;
	ref_gm_rotary 	: ref_sv_io;
	ref_gm_pickUp 	: ref_sv_io;
	ref_gm_stamp 	: ref_sv_io;
END_VAR

// ---- GVLs/gvl_text.TcGVL
{attribute 'qualified_only'}
VAR_GLOBAL
	var_auto_runing: WSTRING(255);
	var_stopping: WSTRING(255);
	var_trayChangeDone: WSTRING(255);
END_VAR

// ---- GVLs/gvl_visu.TcGVL
{attribute 'qualified_only'}
VAR_GLOBAL
	flg_powerOn	: BOOL;
	var_jofAxis : eP_xyz;
	flg_btn_moveDirct : eP_direction;
	flg_btn_PosInit: BOOL;
	flg_btn_PosPickUP: BOOL;
	flg_btn_PosRemove: BOOL;
	flg_btn_PosSample: BOOL;
	flg_btn_PosPocket: BOOL;
	var_in_sampleCavNo: INT := 1;
	var_in_cavNo: INT := 1;
	var_in_pocketNo: INT := 1;
	var_in_samplePos: ref_xyz;
	var_in_initialPos: ref_xyz;
	var_in_removePos: ref_xyz;
	var_in_pickUpPos: ref_xyz;
	var_in_productGenerate: ref_productInfo;
	flg_btn_saveProductInfo: BOOL;
	flg_btn_eleTransportPostive: BOOL;
	flg_btn_eleTransportNegative: BOOL;
	flg_btn_eleSamplePositive: BOOL;
	flg_btn_eleSampleNegative: BOOL;
	flg_btn_eleTrayChangePositive: BOOL;
	flg_btn_eleTrayChangeNegative: BOOL;
	flg_btn_eleRotaryPositive: BOOL;
	flg_btn_eleRotaryNegative: BOOL;
	flg_btn_gm_elePickUpPositive: BOOL;
	flg_btn_gm_elePickUpNegative: BOOL;
	flg_btn_gm_eleTransportPositive: BOOL;
	flg_btn_gm_eleTransportNegative: BOOL;
	flg_btn_svChuckOpen: BOOL;
	flg_btn_svChuckClose: BOOL;
	flg_btn_svPushClose: BOOL;
	flg_btn_svPushOpen: BOOL;
	flg_btn_gm_svChuckOpen: BOOL;
	flg_btn_gm_svChuckClose: BOOL;
	flg_btn_gm_svPushClose: BOOL;
	flg_btn_gm_svPushOpen: BOOL;
	flg_btn_gm_svRotaryOrigin: BOOL;
	flg_btn_gm_svRotaryMoving: BOOL;
	flg_btn_gm_svPickUpOrigin: BOOL;
	flg_btn_gm_svPickUpMoving: BOOL;
	flg_btn_gm_svStampOrigin: BOOL;
	flg_btn_gm_svStampMoving: BOOL;
	flg_btn_vacuumOn: BOOL;
	flg_btn_vacuumOff: BOOL;
	flg_btn_breakOn: BOOL;
	flg_btn_gm_vacuumOn: BOOL;
	flg_btn_gm_vacuumOff: BOOL;
	flg_btn_gm_breakOn: BOOL;
	flg_btn_savePalletize: BOOL;
	flg_btn_saveSample: BOOL;
	flg_btn_sample: BOOL;
	flg_btn_autoModeStop: BOOL;
	flg_btn_gm_motorPower: BOOL;
	flg_btn_vacSensOn: BOOL;
	flg_btn_vacRobotOn: BOOL;
	flg_btn_lensSetDone: BOOL;
	var_DT: DT;
	flg_btn_clrDefectiveQty: BOOL;
	flg_btn_autoModeStart: BOOL;
	flg_btn_trayChangeDone: BOOL;
	var_msg: WSTRING;
	var_dev_passingPosY: LREAL;
	var_dev_passingPosX: LREAL;
	var_dev_passingPosZ: LREAL;
	var_dev_settingPosX: LREAL;
	var_dev_settingPosY: LREAL;
	var_dev_settingPosZ: LREAL;
	var_in_teachingDetail: ref_teachingDetail;
	var_gm_rotaryInch: LREAL;
	flg_btn_rotaryRigt: BOOL;
	flg_btn_rotaryLeft: BOOL;
	var_radio_rotaryJogMode: INT;
	flg_btn_clrPockertQty: BOOL;
	var_rotaryPos: s_gm_rotaryPos;
	flg_btn_rotaryPos: BOOL;
	flg_btn_gm_moveOrigin: BOOL;
	flg_btn_gm_movePickUp: BOOL;
	flg_btn_gm_moveSet: BOOL;
	flg_btn_gm_moveRemove: BOOL;
	var_in_teachingDetailVels: s_velsXYZ;
	var_currentTableMsg : WSTRING;
	var_curenntGateData: LREAL;
	flg_btn_projectReset: BOOL;
	flg_btn_invalidBuzzer: BOOL;
	flg_btn_gateMeasurementPreset: BOOL;
	var_projectResetLastTime: LREAL;
	flg_btn_clrGateData: BOOL;
	flg_btn_buzzer_silent: BOOL;
	flg_btn_All_PosPocket: BOOL;
	flg_All_PosPorket_Move: BOOL;
END_VAR
VAR_GLOBAL PERSISTENT
	var_in_palletizePos: ref_palletize;
	var_radio_jogMode: INT;
	var_in_inch: LREAL:=0.2;
	var_in_currentProduct : ARRAY[0..10] OF STRING;
	flg_btn_usingMeasurementSystem : BOOL;
	flg_btn_gateMeasurementIsNone: BOOL;
	var_dev_palletizingMode: BOOL;
	var_gm_manualRotaryVel: LREAL;
	var_gm_autoRotaryVel: LREAL;
	var_gm_autoRotaryAcc: LREAL;
	var_gm_autoRotaryDec: LREAL;
	var_gateLengthList: ARRAY[0..49] OF REAL;
	var_gateLengthListCav: ARRAY[1..8] OF ARRAY[0..49] OF REAL;
	flg_btn_rotaryReversal: BOOL;
	flg_btn_RotaryIsNotUse: BOOL;
	flg_missingParts: BOOL;
	flg_usingTimeStamp : BOOL;
	var_enableSchedule: ARRAY[0..6] OF BOOL;
	var_scheduleTimeH : ARRAY[0..6] OF WORD;
	var_scheduleTimeM : ARRAY[0..6] OF WORD;
END_VAR

// ---- POUs/MAIN.TcPOU
PROGRAM MAIN
VAR
	fbi_lsm_main: fb_lsm_main;
	fbi_text_control_run: fb_text_control;
END_VAR

fbi_lsm_main();
fbi_text_control_run();

END_PROGRAM

// ---- FBs/fb_lsm_main.TcPOU
FUNCTION_BLOCK fb_lsm_main
VAR_INPUT
END_VAR
VAR_OUTPUT
END_VAR
VAR
	fbi_mapping			:fb_mapping;
	fbi_IO				:fb_IO;
	fbi_modeController	:fb_modeController;
	fbi_motorController	:fb_motorController;
	fbi_eventController	:fb_eventController;
	fbi_eleControllers	:fb_eleControllers;
	fbi_svControllers	:fb_svControllers;
	fbi_recordingSystem :fb_recordingSystem;
	fbi_GetLocalAmsNetId: FB_GetLocalAmsNetId;
	fbi_LocalSystemTime: FB_LocalSystemTime;
	fbi_resetDelay: TON;
	fb_Shutdown: NT_Shutdown;
	fb_Reboot: NT_Reboot;
	ShutdownStart: BOOL;
	RebootStart: BOOL;
	fbi_WritePersistentData: FB_WritePersistentData;
	var_lastTIme: LREAL;
	gvl_error_reset: BOOL;
	fbi_productGenerater: fb_productGenerator;
	fbi_sampleSchedule: fb_sampleSchedule;
	test_flg: BOOL;
END_VAR

THIS^.fbi_mapping();
THIS^.fbi_IO();
THIS^.fbi_modeController();
THIS^.fbi_eleControllers();
THIS^.fbi_svControllers();
THIS^.fbi_recordingSystem();
THIS^.fbi_productGenerater();
THIS^.fbi_motorController();
THIS^.fbi_eventController(in_flg_run:=TRUE , out_flg_run=> );
THIS^.fbi_modeController.p_init := fbi_resetDelay.Q ;
gvl_axis.fbi_motionControler.p_Init := gvl_param.var_currentMode = eP_programMode.error;
fbi_resetDelay(IN:= gvl_visu.flg_btn_projectReset , PT:=T#5S , Q=> , ET=>  );
gvl_visu.var_projectResetLastTime :=(LREAL#5000 - TIME_TO_LREAL(fbi_resetDelay.ET))/1000;
gvl_axis.fbi_motionControler(
	in_flg_run:= TRUE, 
	out_flg_run=> , 
	var_ref_X:= gvl_axis.ref_x, 
	var_ref_Y:= gvl_axis.ref_y, 
	var_ref_Z:= gvl_axis.ref_z, 
	in_flg_start:= gvl_axis.fbi_motionControler.in_flg_start, 
	in_var_targetPosX:= , 
	in_var_targetPosY:= , 
	in_var_targetPosZ:= , 
	in_var_direction:= , 
	out_flg_busy=> , 
	out_flg_Done=> , 
	out_flg_moveXYDone=> );
fbi_sampleSchedule(in_var_enableSchedule:= gvl_visu.var_enableSchedule ,
	in_var_scheduleTimeH:= gvl_visu.var_scheduleTimeH ,
	in_var_scheduleTimeM:= gvl_visu.var_scheduleTimeM ,
	out_flg_sampletriger=> );
	IF fbi_sampleSchedule.out_flg_sampletriger AND gvl_param.var_currentMode = eP_programMode.auto THEN
		gvl_visu.flg_btn_sample := TRUE;
	END_IF
fbi_GetLocalAmsNetId(
	bExecute:=TRUE , 
	tTimeOut:= ,
	bBusy=> , 
	bError=> , 
	nErrId=> , 
	AddrString=> , 
	AddrBytes=> );
fbi_LocalSystemTime(
	sNetID:=fbi_GetLocalAmsNetId.AddrString , 
	bEnable:= TRUE, 
	dwCycle:= , 
	dwOpt:= , 
	tTimeout:= , 
	bValid=> , 
	systemTime=> , 
	tzID=> );
fb_Shutdown(
	NETID:= fbi_GetLocalAmsNetId.AddrString, 
	DELAY:= 3, 
	START:= ShutdownStart, 
	TMOUT:= T#6S, 
	BUSY=> , 
	ERR=> , 
	ERRID=> );

fb_Reboot(
	NETID:= fbi_GetLocalAmsNetId.AddrString, 
	DELAY:= 3, 
	START:= RebootStart, 
	TMOUT:= T#6S, 
	BUSY=> , 
	ERR=> , 
	ERRID=> );
fbi_WritePersistentData(
	NETID:= fbi_GetLocalAmsNetId.AddrString, 
	PORT:= 851, 
	START:= gvl_axis.fbi_motionControler.out_flg_Done, 
	TMOUT:= , 
	MODE:= , 
	BUSY=> , 
	ERR=> , 
	ERRID=> );
gvl_visu.var_DT := SYSTEMTIME_TO_DT(fbi_LocalSystemTime.systemTime);
gvl_visu.var_curenntGateData := DINT_TO_LREAL(gvl_io.var_gateLength)/10000;

END_FUNCTION_BLOCK

// ---- FBs/fb_mapping.TcPOU
FUNCTION_BLOCK fb_mapping
VAR_INPUT
END_VAR
VAR_OUTPUT
END_VAR
VAR
	fbi_ejector_io: ARRAY[1..3] OF fb_ejector_io;
	fbi_sv_io: ARRAY[1..8] OF  fb_sv_io;
	fbi_ele_io: ARRAY[1..6] OF  fb_ele_io;
END_VAR

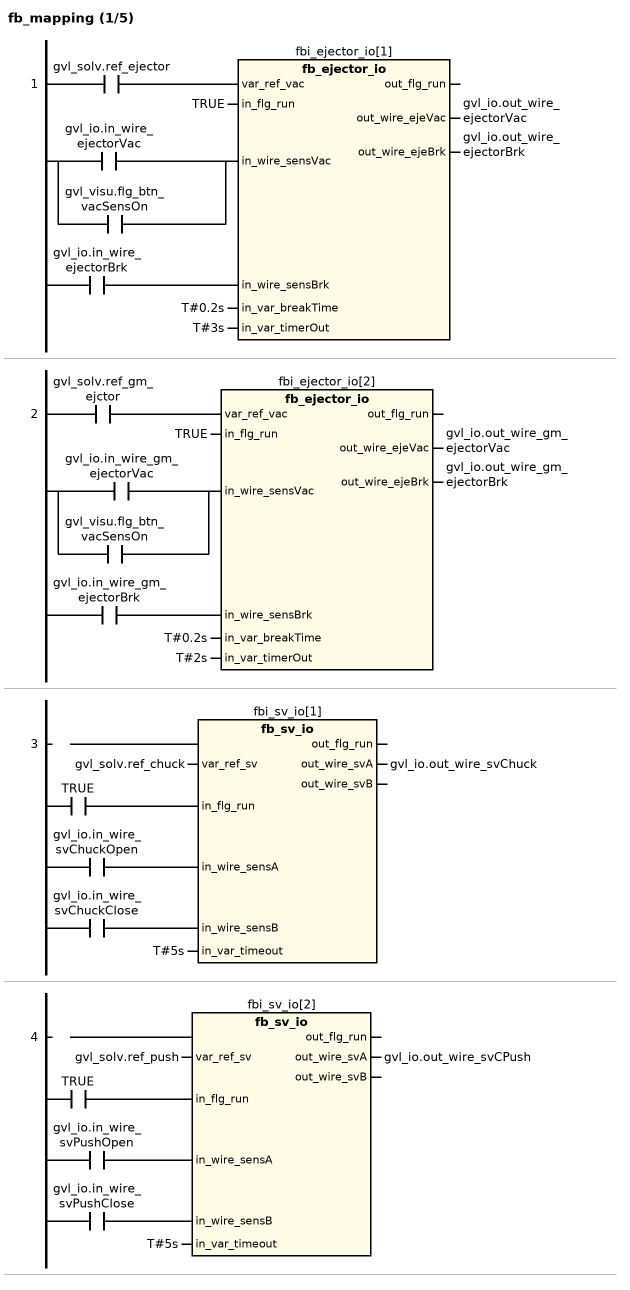
// NETWORK 1
fbi_ejector_io[1](
    var_ref_vac := gvl_solv.ref_ejector,
    in_flg_run := TRUE,
    in_wire_sensVac := gvl_io.in_wire_ejectorVac OR gvl_visu.flg_btn_vacSensOn,
    in_wire_sensBrk := gvl_io.in_wire_ejectorBrk,
    in_var_breakTime := T#0.2s,
    in_var_timerOut := T#3s,
    out_wire_ejeVac => gvl_io.out_wire_ejectorVac,
    out_wire_ejeBrk => gvl_io.out_wire_ejectorBrk); // fb_ejector_io

// NETWORK 2
fbi_ejector_io[2](
    var_ref_vac := gvl_solv.ref_gm_ejctor,
    in_flg_run := TRUE,
    in_wire_sensVac := gvl_io.in_wire_gm_ejectorVac OR gvl_visu.flg_btn_vacSensOn,
    in_wire_sensBrk := gvl_io.in_wire_gm_ejectorBrk,
    in_var_breakTime := T#0.2s,
    in_var_timerOut := T#2s,
    out_wire_ejeVac => gvl_io.out_wire_gm_ejectorVac,
    out_wire_ejeBrk => gvl_io.out_wire_gm_ejectorBrk); // fb_ejector_io

// NETWORK 3
fbi_sv_io[1](
    var_ref_sv := gvl_solv.ref_chuck,
    in_flg_run := TRUE,
    in_wire_sensA := gvl_io.in_wire_svChuckOpen,
    in_wire_sensB := gvl_io.in_wire_svChuckClose,
    in_var_timeout := T#5s,
    out_wire_svA => gvl_io.out_wire_svChuck); // fb_sv_io

// NETWORK 4
fbi_sv_io[2](
    var_ref_sv := gvl_solv.ref_push,
    in_flg_run := TRUE,
    in_wire_sensA := gvl_io.in_wire_svPushOpen,
    in_wire_sensB := gvl_io.in_wire_svPushClose,
    in_var_timeout := T#5s,
    out_wire_svA => gvl_io.out_wire_svCPush); // fb_sv_io

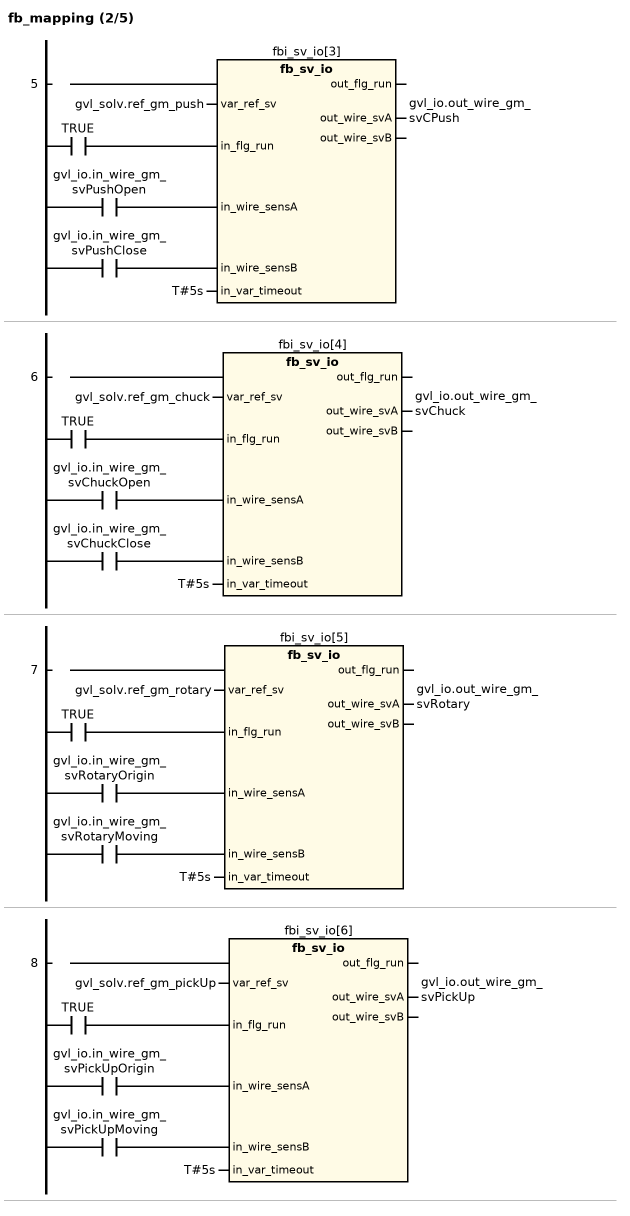
// NETWORK 5
fbi_sv_io[3](
    var_ref_sv := gvl_solv.ref_gm_push,
    in_flg_run := TRUE,
    in_wire_sensA := gvl_io.in_wire_gm_svPushOpen,
    in_wire_sensB := gvl_io.in_wire_gm_svPushClose,
    in_var_timeout := T#5s,
    out_wire_svA => gvl_io.out_wire_gm_svCPush); // fb_sv_io

// NETWORK 6
fbi_sv_io[4](
    var_ref_sv := gvl_solv.ref_gm_chuck,
    in_flg_run := TRUE,
    in_wire_sensA := gvl_io.in_wire_gm_svChuckOpen,
    in_wire_sensB := gvl_io.in_wire_gm_svChuckClose,
    in_var_timeout := T#5s,
    out_wire_svA => gvl_io.out_wire_gm_svChuck); // fb_sv_io

// NETWORK 7
fbi_sv_io[5](
    var_ref_sv := gvl_solv.ref_gm_rotary,
    in_flg_run := TRUE,
    in_wire_sensA := gvl_io.in_wire_gm_svRotaryOrigin,
    in_wire_sensB := gvl_io.in_wire_gm_svRotaryMoving,
    in_var_timeout := T#5s,
    out_wire_svA => gvl_io.out_wire_gm_svRotary); // fb_sv_io

// NETWORK 8
fbi_sv_io[6](
    var_ref_sv := gvl_solv.ref_gm_pickUp,
    in_flg_run := TRUE,
    in_wire_sensA := gvl_io.in_wire_gm_svPickUpOrigin,
    in_wire_sensB := gvl_io.in_wire_gm_svPickUpMoving,
    in_var_timeout := T#5s,
    out_wire_svA => gvl_io.out_wire_gm_svPickUp); // fb_sv_io

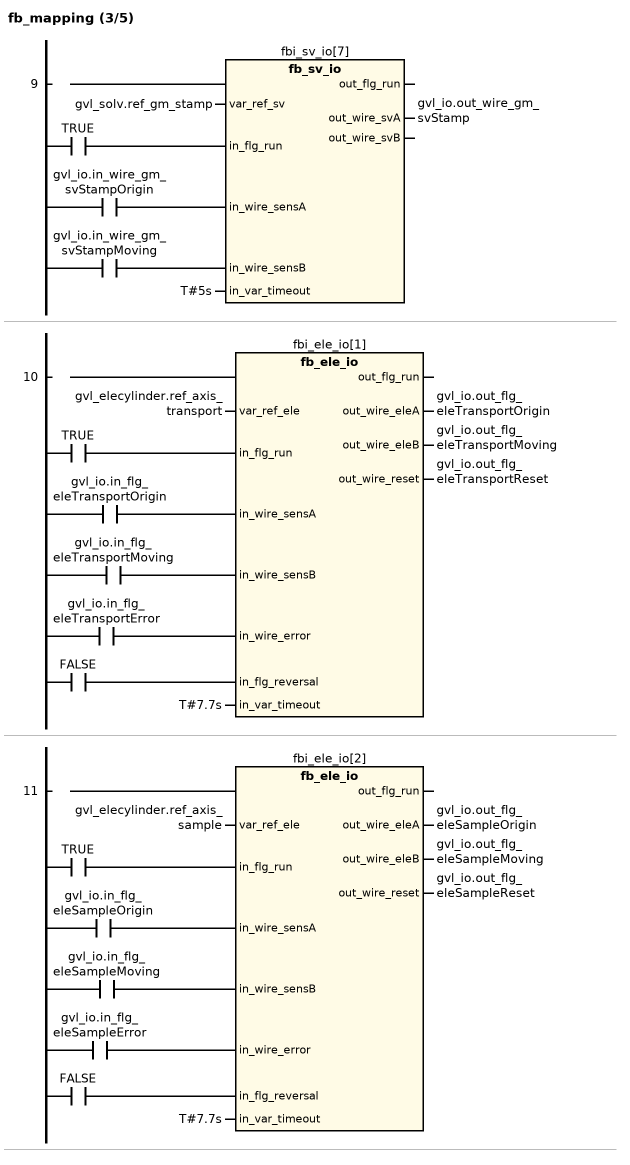
// NETWORK 9
fbi_sv_io[7](
    var_ref_sv := gvl_solv.ref_gm_stamp,
    in_flg_run := TRUE,
    in_wire_sensA := gvl_io.in_wire_gm_svStampOrigin,
    in_wire_sensB := gvl_io.in_wire_gm_svStampMoving,
    in_var_timeout := T#5s,
    out_wire_svA => gvl_io.out_wire_gm_svStamp); // fb_sv_io

// NETWORK 10
fbi_ele_io[1](
    var_ref_ele := gvl_elecylinder.ref_axis_transport,
    in_flg_run := TRUE,
    in_wire_sensA := gvl_io.in_flg_eleTransportOrigin,
    in_wire_sensB := gvl_io.in_flg_eleTransportMoving,
    in_wire_error := gvl_io.in_flg_eleTransportError,
    in_flg_reversal := FALSE,
    in_var_timeout := T#7.7s,
    out_wire_eleA => gvl_io.out_flg_eleTransportOrigin,
    out_wire_eleB => gvl_io.out_flg_eleTransportMoving,
    out_wire_reset => gvl_io.out_flg_eleTransportReset); // fb_ele_io

// NETWORK 11
fbi_ele_io[2](
    var_ref_ele := gvl_elecylinder.ref_axis_sample,
    in_flg_run := TRUE,
    in_wire_sensA := gvl_io.in_flg_eleSampleOrigin,
    in_wire_sensB := gvl_io.in_flg_eleSampleMoving,
    in_wire_error := gvl_io.in_flg_eleSampleError,
    in_flg_reversal := FALSE,
    in_var_timeout := T#7.7s,
    out_wire_eleA => gvl_io.out_flg_eleSampleOrigin,
    out_wire_eleB => gvl_io.out_flg_eleSampleMoving,
    out_wire_reset => gvl_io.out_flg_eleSampleReset); // fb_ele_io

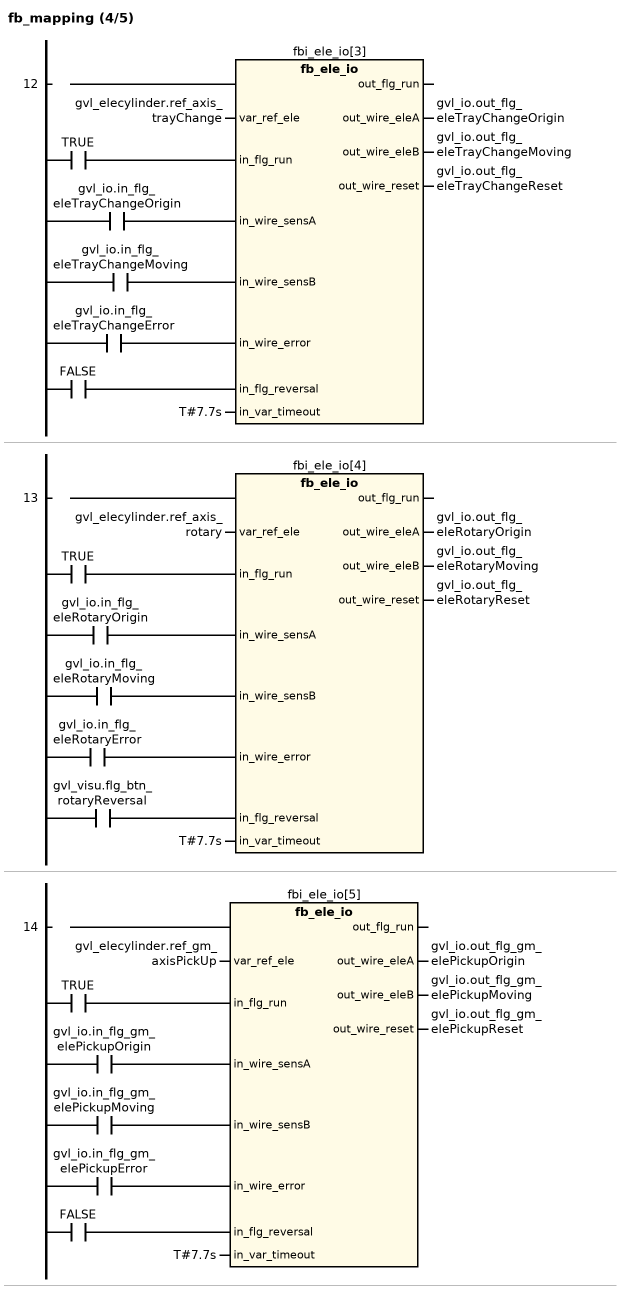
// NETWORK 12
fbi_ele_io[3](
    var_ref_ele := gvl_elecylinder.ref_axis_trayChange,
    in_flg_run := TRUE,
    in_wire_sensA := gvl_io.in_flg_eleTrayChangeOrigin,
    in_wire_sensB := gvl_io.in_flg_eleTrayChangeMoving,
    in_wire_error := gvl_io.in_flg_eleTrayChangeError,
    in_flg_reversal := FALSE,
    in_var_timeout := T#7.7s,
    out_wire_eleA => gvl_io.out_flg_eleTrayChangeOrigin,
    out_wire_eleB => gvl_io.out_flg_eleTrayChangeMoving,
    out_wire_reset => gvl_io.out_flg_eleTrayChangeReset); // fb_ele_io

// NETWORK 13
fbi_ele_io[4](
    var_ref_ele := gvl_elecylinder.ref_axis_rotary,
    in_flg_run := TRUE,
    in_wire_sensA := gvl_io.in_flg_eleRotaryOrigin,
    in_wire_sensB := gvl_io.in_flg_eleRotaryMoving,
    in_wire_error := gvl_io.in_flg_eleRotaryError,
    in_flg_reversal := gvl_visu.flg_btn_rotaryReversal,
    in_var_timeout := T#7.7s,
    out_wire_eleA => gvl_io.out_flg_eleRotaryOrigin,
    out_wire_eleB => gvl_io.out_flg_eleRotaryMoving,
    out_wire_reset => gvl_io.out_flg_eleRotaryReset); // fb_ele_io

// NETWORK 14
fbi_ele_io[5](
    var_ref_ele := gvl_elecylinder.ref_gm_axisPickUp,
    in_flg_run := TRUE,
    in_wire_sensA := gvl_io.in_flg_gm_elePickupOrigin,
    in_wire_sensB := gvl_io.in_flg_gm_elePickupMoving,
    in_wire_error := gvl_io.in_flg_gm_elePickupError,
    in_flg_reversal := FALSE,
    in_var_timeout := T#7.7s,
    out_wire_eleA => gvl_io.out_flg_gm_elePickupOrigin,
    out_wire_eleB => gvl_io.out_flg_gm_elePickupMoving,
    out_wire_reset => gvl_io.out_flg_gm_elePickupReset); // fb_ele_io

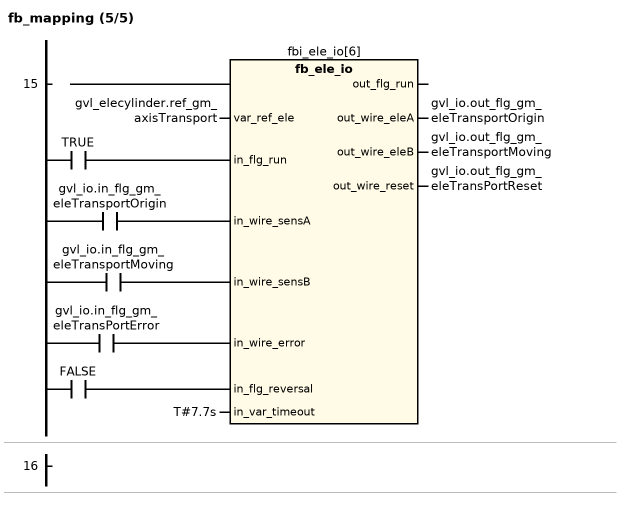
// NETWORK 15
fbi_ele_io[6](
    var_ref_ele := gvl_elecylinder.ref_gm_axisTransport,
    in_flg_run := TRUE,
    in_wire_sensA := gvl_io.in_flg_gm_eleTransportOrigin,
    in_wire_sensB := gvl_io.in_flg_gm_eleTransportMoving,
    in_wire_error := gvl_io.in_flg_gm_eleTransPortError,
    in_flg_reversal := FALSE,
    in_var_timeout := T#7.7s,
    out_wire_eleA => gvl_io.out_flg_gm_eleTransportOrigin,
    out_wire_eleB => gvl_io.out_flg_gm_eleTransportMoving,
    out_wire_reset => gvl_io.out_flg_gm_eleTransPortReset); // fb_ele_io

// NETWORK 16

END_FUNCTION_BLOCK

// ---- FBs/fb_ejecter/fb_ejector_io.TcPOU
FUNCTION_BLOCK fb_ejector_io
VAR_IN_OUT
	var_ref_vac : ref_eje_io;
END_VAR
VAR_INPUT
	in_flg_run : BOOL;
	in_wire_sensVac : BOOL;
	in_wire_sensBrk : BOOL;
	in_var_breakTime: TIME;
	in_var_timerOut : TIME;
END_VAR
VAR_OUTPUT
	out_flg_run : BOOL;
	out_wire_ejeVac : BOOL;
	out_wire_ejeBrk : BOOL;
END_VAR
VAR
END_VAR

out_flg_run := in_flg_run;

var_ref_vac.input.in_flg_sensVac := in_wire_sensVac;
var_ref_vac.input.in_flg_sensBrk := in_wire_sensBrk;

out_wire_ejeVac := var_ref_vac.output.out_flg_ejeVac;
out_wire_ejeBrk := var_ref_vac.output.out_flg_ejeBrk;

var_ref_vac.param.var_BrkTime := in_var_breakTime;
var_ref_vac.param.var_timeOut := in_var_timerOut;

END_FUNCTION_BLOCK

// ---- FBs/fb_sv/fb_sv_io.TcPOU
FUNCTION_BLOCK fb_sv_io
VAR_IN_OUT
	var_ref_sv : ref_sv_io;
END_VAR
VAR_INPUT
	in_flg_run : BOOL;
	in_wire_sensA : BOOL;
	in_wire_sensB : BOOL;
	in_var_timeout : time;
END_VAR
VAR_OUTPUT
	out_flg_run : BOOL;
	out_wire_svA : BOOL;
	out_wire_svB : BOOL;
END_VAR
VAR
END_VAR

out_flg_run := in_flg_run;
var_ref_sv.in.in_flg_sensA := in_wire_sensA;
var_ref_sv.in.in_flg_sensB := in_wire_sensB;

IF var_ref_sv.param.var_svType = eP_svType.single THEN
	out_wire_svA := var_ref_sv.out.out_flg_svA;
	out_wire_svB := var_ref_sv.out.out_flg_svB;
ELSIF var_ref_sv.param.var_svType = eP_svType.double THEN
	IF var_ref_sv.out.out_flg_svA THEN
		IF var_ref_sv.in.in_flg_sensA THEN
			out_wire_svA := FALSE;
		ELSE
			out_wire_svA := TRUE;
		END_IF
	ELSIF var_ref_sv.out.out_flg_svB THEN
		IF var_ref_sv.in.in_flg_sensB THEN
			out_wire_svB := FALSE;
		ELSE
			out_wire_svB := TRUE;
		END_IF
	END_IF
END_IF
var_ref_sv.param.var_timeOut := in_var_timeout;

END_FUNCTION_BLOCK

// ---- FBs/fb_ele/fb_ele_io.TcPOU
FUNCTION_BLOCK fb_ele_io
VAR_IN_OUT
	var_ref_ele : ref_ele_io;
END_VAR
VAR_INPUT
	in_flg_run : BOOL;
	in_wire_sensA : BOOL;
	in_wire_sensB : BOOL;
	in_wire_error : BOOL;
	in_flg_reversal: BOOL;
	in_var_timeout : TIME;
END_VAR
VAR_OUTPUT
	out_flg_run : BOOL;
	out_wire_eleA : BOOL;
	out_wire_eleB : BOOL;
	out_wire_reset : BOOL;

END_VAR
VAR
END_VAR

out_flg_run := in_flg_run;
IF in_flg_reversal THEN
	var_ref_ele.input.in_flg_sensA := in_wire_sensB;
	var_ref_ele.input.in_flg_sensB := in_wire_sensA;
	var_ref_ele.input.in_wire_error := NOT in_wire_error;
	
	out_wire_eleA := var_ref_ele.output.out_flg_eleB;
	out_wire_eleB := var_ref_ele.output.out_flg_eleA;
	out_wire_reset := var_ref_ele.output.out_flg_reset;
ELSE
	var_ref_ele.input.in_flg_sensA := in_wire_sensA;
	var_ref_ele.input.in_flg_sensB := in_wire_sensB;
	var_ref_ele.input.in_wire_error := NOT in_wire_error;
	
	out_wire_eleA := var_ref_ele.output.out_flg_eleA;
	out_wire_eleB := var_ref_ele.output.out_flg_eleB;
	out_wire_reset := var_ref_ele.output.out_flg_reset;
END_IF

IF in_wire_sensA = FALSE AND in_wire_sensB = FALSE THEN
	var_ref_ele.input.in_flg_sensNone := TRUE;
ELSE
	var_ref_ele.input.in_flg_sensNone := FALSE;
END_IF
var_ref_ele.param.var_timeOut := in_var_timeout;

END_FUNCTION_BLOCK

// ---- FBs/fb_IO.TcPOU
FUNCTION_BLOCK fb_IO
VAR_INPUT
END_VAR
VAR_OUTPUT
END_VAR
VAR
	fbi_incjetMapping :	fb_incjetMapping;
END_VAR

gvl_io.flg_bitNumber0 					:= gvl_io.in_bitNumber0;
gvl_io.flg_bitNumber1 					:= gvl_io.in_bitNumber1;
gvl_io.flg_bitNumber2 					:= gvl_io.in_bitNumber2;
gvl_io.flg_bitNumber3 					:= gvl_io.in_bitNumber3;
gvl_io.flg_dummySiganl 					:= gvl_io.in_wire_dummySignal;
gvl_io.flg_gateLengthIsSuccessed 		:= gvl_io.in_wire_gatelengthIsSuccessed;
gvl_io.flg_lensSetDone 					:= gvl_io.in_wire_lensSetDone;
gvl_io.flg_fiberSens 					:= gvl_io.in_wire_fiberSens;
gvl_io.flg_btnGreen 					:= gvl_io.in_wire_btnGreen;
gvl_io.flg_btnRed 						:= gvl_io.in_wire_btnRed;
gvl_io.flg_frontSaftyDoor 				:= gvl_io.in_wire_frontSaftyDoor;
gvl_io.var_gateLength 					:= gvl_io.in_wire_gateLength;
gvl_io.flg_gatemeasurementStatus 		:= gvl_io.in_wire_gateMeasurementStatus;
gvl_io.var_gateMeasurementErrCode.0		:= gvl_io.in_wire_gateMeasurementErrCode.0;
gvl_io.var_gateMeasurementErrCode.1		:= gvl_io.in_wire_gateMeasurementErrCode.1;
gvl_io.out_wire_gateMeasurementReset	:=	gvl_io.var_gateMeasurementReset	;
gvl_io.out_wire_gateMeasurementPreset	:=	gvl_io.var_gateMeasurementPreset;
gvl_io.flg_gm_fiberSens 				:= gvl_io.in_wire_gm_fiberSens;
gvl_io.flg_saftyUnitState 				:= gvl_io.in_wire_saftyUnitState;

gvl_io.out_wire_saftyUnitReset 			:= gvl_io.flg_saftyUnitReset;
gvl_io.out_wire_requestLens 			:= gvl_io.flg_requestLens;
gvl_io.out_wire_signalTowerBuzzer 		:= gvl_io.flg_signalTowerBuzzer AND NOT gvl_visu.flg_btn_invalidBuzzer;
gvl_io.out_wire_signalTowerGreen 		:= gvl_io.flg_signalTowerGreen;
gvl_io.out_wire_signalTowerRed 			:= gvl_io.flg_signalTowerRed;
gvl_io.out_wire_signalTowerYellow 		:= gvl_io.flg_signalTowerYellow;

//elecylinder

gvl_io.in_flg_eleTransportOrigin 		:= gvl_io.in_wire_ele_stocker.0;
gvl_io.in_flg_eleTransportMoving 		:= gvl_io.in_wire_ele_stocker.1;
gvl_io.in_flg_eleTransportError 		:= gvl_io.in_wire_ele_stocker.2;
gvl_io.in_flg_eleRotaryOrigin			:= gvl_io.in_wire_ele_stocker.4;
gvl_io.in_flg_eleRotaryMoving			:= gvl_io.in_wire_ele_stocker.5;
gvl_io.in_flg_eleRotaryError			:= gvl_io.in_wire_ele_stocker.6;
gvl_io.in_flg_eleSampleOrigin			:= gvl_io.in_wire_ele_stocker.8;
gvl_io.in_flg_eleSampleMoving			:= gvl_io.in_wire_ele_stocker.9;
gvl_io.in_flg_eleSampleError			:= gvl_io.in_wire_ele_stocker.10;
gvl_io.in_flg_eleTrayChangeOrigin		:= gvl_io.in_wire_ele_stocker.12;
gvl_io.in_flg_eleTrayChangeMoving		:= gvl_io.in_wire_ele_stocker.13;
gvl_io.in_flg_eleTrayChangeError		:= gvl_io.in_wire_ele_stocker.14;
gvl_io.in_flg_gm_eleTransportOrigin		:= gvl_io.in_wire_ele_gateMeasurement.0;
gvl_io.in_flg_gm_eleTransportMoving		:= gvl_io.in_wire_ele_gateMeasurement.1;
gvl_io.in_flg_gm_eleTransPortError		:= gvl_io.in_wire_ele_gateMeasurement.2;
gvl_io.in_flg_gm_elePickupOrigin		:= gvl_io.in_wire_ele_gateMeasurement.5;
gvl_io.in_flg_gm_elePickupMoving		:= gvl_io.in_wire_ele_gateMeasurement.4;
gvl_io.in_flg_gm_elePickupError			:= gvl_io.in_wire_ele_gateMeasurement.6;

gvl_io.out_wire_ele_stocker.0			:= gvl_io.out_flg_eleTransportOrigin;
gvl_io.out_wire_ele_stocker.1			:= gvl_io.out_flg_eleTransportMoving;
gvl_io.out_wire_ele_stocker.2			:= gvl_io.out_flg_eleTransportReset;
gvl_io.out_wire_ele_stocker.4			:= gvl_io.out_flg_eleRotaryOrigin;
gvl_io.out_wire_ele_stocker.5			:= gvl_io.out_flg_eleRotaryMoving;
gvl_io.out_wire_ele_stocker.6			:= gvl_io.out_flg_eleRotaryReset;
gvl_io.out_wire_ele_stocker.8			:= gvl_io.out_flg_eleSampleOrigin;
gvl_io.out_wire_ele_stocker.9			:= gvl_io.out_flg_eleSampleMoving;
gvl_io.out_wire_ele_stocker.10			:= gvl_io.out_flg_eleSampleReset;
gvl_io.out_wire_ele_stocker.12			:= gvl_io.out_flg_eleTrayChangeOrigin;
gvl_io.out_wire_ele_stocker.13			:= gvl_io.out_flg_eleTrayChangeMoving;
gvl_io.out_wire_ele_stocker.14			:= gvl_io.out_flg_eleTrayChangeReset;
gvl_io.out_wire_ele_gateMeasurement.0 	:= gvl_io.out_flg_gm_eleTransportOrigin;
gvl_io.out_wire_ele_gateMeasurement.1 	:= gvl_io.out_flg_gm_eleTransportMoving;
gvl_io.out_wire_ele_gateMeasurement.2 	:= gvl_io.out_flg_gm_eleTransPortReset;
gvl_io.out_wire_ele_gateMeasurement.5 	:= gvl_io.out_flg_gm_elePickupOrigin;
gvl_io.out_wire_ele_gateMeasurement.4 	:= gvl_io.out_flg_gm_elePickupMoving;
gvl_io.out_wire_ele_gateMeasurement.6 	:= gvl_io.out_flg_gm_elePickupReset;


fbi_incjetMapping(
	IN_00:= gvl_io.in_wire_incjet_error, 
	IN_01:= , 
	IN_02:= , 
	IN_03:= gvl_io.in_wire_incjet_ready, 
	IN_04:= , 
	IN_05:= , 
	IN_06:= gvl_io.in_wire_incjet_run,
	IN_07:= , 
	IN_08:= , 
	IN_09:= , 
	OUT_00=> , 
	OUT_01=> , 
	OUT_02=> , 
	OUT_03=> , 
	OUT_04=> , 
	OUT_05=> , 
	OUT_06=> , 
	OUT_07=> , 
	OUT_08=> gvl_io.out_wire_incjet_stampDeny, 
	OUT_09=> , 
	OUT_10=> , 
	OUT_11=> , 
	OUT_12=> , 
	OUT_13=> , 
	OUT_14=> , 
	OUT_15=> , 
	OUT_16=> , 
	OUT_17=> , 
	OUT_18=> , 
	OUT_19=> , 
	var_productInfo:= gvl_param.var_productInfo[gvl_param.var_currentProductID], 
	var_incjetInfo:= gvl_gm.var_incjetInfo);

END_FUNCTION_BLOCK

// ---- FBs/Incjet/fb_incjetMapping.TcPOU
FUNCTION_BLOCK fb_incjetMapping
VAR_INPUT
	IN_00 : BOOL;
	IN_01 : BOOL;
	IN_02 : BOOL;
	IN_03 : BOOL;
	IN_04 : BOOL;
	IN_05 : BOOL;
	IN_06 : BOOL;
	IN_07 : BOOL;
	IN_08 : BOOL;
	IN_09 : BOOL;
END_VAR
VAR_OUTPUT
	OUT_00 : BOOL;
	OUT_01 : BOOL;
	OUT_02 : BOOL;
	OUT_03 : BOOL;
	OUT_04 : BOOL;
	OUT_05 : BOOL;
	OUT_06 : BOOL;
	OUT_07 : BOOL;
	OUT_08 : BOOL;
	OUT_09 : BOOL;
	OUT_10 : BOOL;
	OUT_11 : BOOL;
	OUT_12 : BOOL;
	OUT_13 : BOOL;
	OUT_14 : BOOL;
	OUT_15 : BOOL;
	OUT_16 : BOOL;
	OUT_17 : BOOL;
	OUT_18 : BOOL;
	OUT_19 : BOOL;
END_VAR
VAR_IN_OUT
	var_productInfo : ref_productInfo;
	var_incjetInfo : ref_incjetInfo;
END_VAR
VAR
END_VAR

var_incjetInfo.var_msgNo := var_productInfo.incjetMsgNo;
OUT_00 := var_incjetInfo.var_msgNo.0;
OUT_01 := var_incjetInfo.var_msgNo.1;
OUT_02 := var_incjetInfo.var_msgNo.2;
OUT_03 := var_incjetInfo.var_msgNo.3;
OUT_04 := var_incjetInfo.var_msgNo.4;
OUT_05 := var_incjetInfo.var_msgNo.5;
OUT_06 := var_incjetInfo.var_msgNo.6;
OUT_07 := var_incjetInfo.var_msgNo.7;

OUT_08 := var_incjetInfo.flg_denyStamp;
//OUT_09  (stop Calendar update)
OUT_10 := var_incjetInfo.flg_numberingCount;
OUT_11 := var_incjetInfo.flg_numberingStop;
OUT_12 := var_incjetInfo.flg_numberingReset;
//OUT_13 :=
//OUT_14 :=
//OUT_15 :=
//OUT_16 := msg no
//OUT_17 := msg no
//OUT_18 := msg no
//OUT_19 := msg no

var_incjetInfo.flg_error := gvl_visu.flg_usingTimeStamp AND IN_00;
var_incjetInfo.flg_incFluxLow := gvl_visu.flg_usingTimeStamp AND IN_01;
var_incjetInfo.flg_stampReady := gvl_visu.flg_usingTimeStamp AND (IN_03 OR (gvl_debug.flg_stampReady AND gvl_debug.flg_debug_run));
var_incjetInfo.flg_stampDone := gvl_visu.flg_usingTimeStamp AND (IN_04 OR (gvl_debug.flg_stampDone AND gvl_debug.flg_debug_run));
var_incjetInfo.flg_stampRun := gvl_visu.flg_usingTimeStamp AND IN_06;

END_FUNCTION_BLOCK

// ---- FBs/fb_modeController.TcPOU
FUNCTION_BLOCK fb_modeController
VAR_INPUT
END_VAR
VAR_OUTPUT
END_VAR
VAR
	SFCInit : BOOL;
	trn_autoRun: BOOL;
	fbi_manual: fb_manual;
	fbi_auto: fb_auto;
	fbi_paramInit: fb_paramInit;	
	trn_autoDone: BOOL;
	var_process: INT;
	fbi_delayTimer0: TON;
	fbi_delayTimer1: TON;
	fbi_delayTimer2: TON;
	fbi_delayTimer3: TON;
	MC_ResetX: MC_Reset;
	MC_ResetY: MC_Reset;
	MC_ResetZ: MC_Reset;
	trn_SaftyUnitResetDone: BOOL;
	resetDelay: TON;
	MC_ResetR: MC_Reset;
	MC_Stop_x: MC_Stop;
	MC_Stop_y: MC_Stop;
	MC_Stop_z: MC_Stop;
	MC_Stop_r: MC_Stop;
	fbi_delayTimer4: TON;
	fbi_timer: TON;
END_VAR
VAR_STAT
	
END_VAR

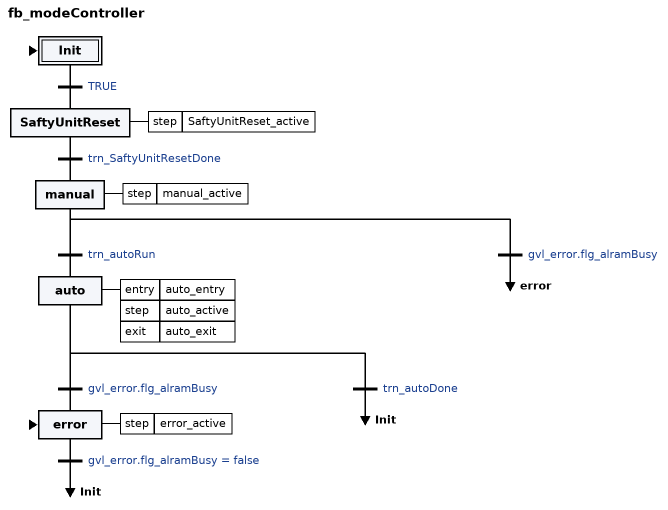
INITIAL_STEP Init:
END_STEP
TRANSITION FROM Init TO SaftyUnitReset
    := TRUE;
END_TRANSITION
STEP SaftyUnitReset:
    SaftyUnitReset_active(N);  // step action
END_STEP
TRANSITION FROM SaftyUnitReset TO manual
    := trn_SaftyUnitResetDone;
END_TRANSITION
STEP manual:
    manual_active(N);  // step action
END_STEP
TRANSITION FROM manual TO auto
    := trn_autoRun;
END_TRANSITION
TRANSITION FROM manual TO error
    := gvl_error.flg_alramBusy;
END_TRANSITION
STEP auto:
    auto_entry(P1);  // entry action
    auto_active(N);  // step action
    auto_exit(P0);  // exit action
END_STEP
TRANSITION FROM auto TO error
    := gvl_error.flg_alramBusy;
END_TRANSITION
TRANSITION FROM auto TO Init
    := trn_autoDone;
END_TRANSITION
STEP error:
    error_active(N);  // step action
END_STEP
TRANSITION FROM error TO Init
    := gvl_error.flg_alramBusy = false;
END_TRANSITION

ACTION auto_active:
IF auto._x AND auto.x = FALSE THEN
	gvl_io.flg_signalTowerGreen := TRUE;
	gvl_io.flg_signalTowerYellow := FALSE;
	gvl_io.flg_signalTowerRed := FALSE;
	trn_autoDone := FALSE;
	THIS^.fbi_auto.p_Init := TRUE;
	THIS^.fbi_auto();
	gvl_auto.requirementToPickUpLens := FALSE;
	gvl_visu.flg_btn_autoModeStop := FALSE;
	gvl_auto.autoModeStoped := FALSE;
	gvl_auto.autoModeStop := FALSE;
	
	gvl_axis.ref_x.Velocity 	:= gvl_param.var_productInfo[gvl_param.var_currentProductID].autoVels.x.vel;
	gvl_axis.ref_x.Acceleration	:= gvl_param.var_productInfo[gvl_param.var_currentProductID].autoVels.x.acc;
	gvl_axis.ref_x.Deceleration	:= gvl_param.var_productInfo[gvl_param.var_currentProductID].autoVels.x.dcc;
	gvl_axis.ref_y.Velocity		:= gvl_param.var_productInfo[gvl_param.var_currentProductID].autoVels.y.vel;
	gvl_axis.ref_y.Acceleration	:= gvl_param.var_productInfo[gvl_param.var_currentProductID].autoVels.y.acc;
	gvl_axis.ref_y.Deceleration	:= gvl_param.var_productInfo[gvl_param.var_currentProductID].autoVels.y.dcc;
	gvl_axis.ref_z.Velocity		:= gvl_param.var_productInfo[gvl_param.var_currentProductID].autoVels.z.vel;
	gvl_axis.ref_z.Acceleration	:= gvl_param.var_productInfo[gvl_param.var_currentProductID].autoVels.z.acc;
	gvl_axis.ref_z.Deceleration	:= gvl_param.var_productInfo[gvl_param.var_currentProductID].autoVels.z.dcc;
	gvl_axis.ref_r.Velocity		:= gvl_gm.var_buf_autoVel;
	gvl_axis.ref_r.Acceleration	:= gvl_gm.var_buf_autoAcc;
	gvl_axis.ref_r.Deceleration	:= gvl_gm.var_buf_autoDec;
	gvl_param.var_currentMode := eP_programMode.auto;
ELSIF auto._x AND auto.x THEN
	gvl_visu.flg_btn_invalidBuzzer := FALSE;
	THIS^.fbi_auto.p_Init := FALSE;
	THIS^.fbi_auto();
	IF gvl_visu.flg_btn_autoModeStop THEN
		gvl_auto.autoModeStop := TRUE;
	END_IF
	IF gvl_auto.autoModeStoped THEN
		trn_autoDone := TRUE;
	END_IF
END_IF
END_ACTION

ACTION auto_entry:
gvl_auto.requirementToPickUpLens := FALSE;
gvl_auto.autoModeStoped := FALSE;
gvl_auto.autoModeStop := FALSE;
gvl_auto.flg_gm_measurementClosed := FALSE;
gvl_auto.flg_gm_transportClosed := FALSE;
gvl_auto.flg_transportClosed := false;
END_ACTION

ACTION auto_exit:
gvl_auto.requirementToPickUpLens := FALSE;
gvl_auto.autoModeStoped := FALSE;
gvl_auto.autoModeStop := FALSE;
gvl_auto.flg_gm_measurementClosed := FALSE;
gvl_auto.flg_gm_transportClosed := FALSE;
gvl_auto.flg_transportClosed := FALSE;
gvl_io.flg_requestLens := FALSE;
gvl_auto.flg_axisIsPcikingUp := FALSE;
gvl_auto.flg_gm_eleIsDown := FALSE;
gvl_visu.flg_btn_sample := FALSE;
gvl_gm.var_incjetInfo.flg_denyStamp := FALSE;
END_ACTION

ACTION error_active:
IF error._x AND error.x = FALSE THEN
	gvl_io.flg_signalTowerGreen := FALSE;
	gvl_io.flg_signalTowerYellow := FALSE;
	gvl_axis.fbi_motionControler.p_Init := TRUE;
	gvl_param.var_currentMode := eP_programMode.error;
	fbi_paramInit.in_flg_run := FALSE;
	fbi_delayTimer0.in := FALSE;
	fbi_delayTimer1.IN := FALSE;
	fbi_delayTimer2.IN := FALSE;
	fbi_delayTimer3.IN := FALSE;
	fbi_delayTimer4.IN := FALSE;
	var_process := 0;
ELSIF error._x AND error.x THEN
	CASE var_process OF
		0:
			MC_Stop_x.Execute := TRUE;
			MC_Stop_y.Execute := TRUE;
			MC_Stop_z.Execute := TRUE;
			IF gvl_visu.flg_btn_usingMeasurementSystem THEN
				MC_Stop_r.Execute := TRUE;
			END_IF
			var_process := 1;
		1:
			MC_Stop_x.Execute := FALSE;
			MC_Stop_y.Execute := FALSE;
			MC_Stop_z.Execute := FALSE;	
			MC_Stop_r.Execute := FALSE;	
			IF gvl_error.flg_reset THEN
				var_process := 2;
			END_IF
		2:
			gvl_io.var_gateMeasurementReset := 0;
			gvl_error.flg_vacuum := FALSE;
			gvl_error.flg_fiberSens := FALSE;
			gvl_error.flg_gm_fiberSens := FALSE;
			gvl_error.flg_incjet := FALSE;
			gvl_error.flg_sample_windown_error:= FALSE;
			gvl_axis.fbi_motionControler.p_Init := FALSE;
			fbi_paramInit.in_flg_run := TRUE;
			gvl_io.var_gateMeasurementReset := 1;
			IF fbi_paramInit.out_flg_done THEN
				fbi_paramInit.in_flg_run := FALSE;
				gvl_visu.var_msg:="";
				var_process := 3;
			END_IF
		3:
			fbi_delayTimer0.IN := TRUE;
			gvl_io.flg_saftyUnitReset := TRUE;
			IF fbi_delayTimer0.Q THEN
				gvl_io.flg_saftyUnitReset := FALSE;
				var_process := 7;
			END_IF
//		4:
//			gvl_elecylinder.fbi_gm_axisTransport.in_flg_run := FALSE;
//			gvl_elecylinder.fbi_gm_axisPickUp.in_flg_run := FALSE;
//			var_process := 5;
//		5:
//			gvl_elecylinder.fbi_gm_axisTransport.in_var_moveMode := eP_eleMoveMode.eleA;
//			gvl_elecylinder.fbi_gm_axisPickUp.in_var_moveMode := eP_eleMoveMode.eleA;
//			gvl_elecylinder.fbi_gm_axisTransport.in_flg_run := TRUE;
//			gvl_elecylinder.fbi_gm_axisPickUp.in_flg_run := TRUE;
//			var_process := 6;
//		6:
//			IF gvl_elecylinder.fbi_gm_axisTransport.out_flg_Done AND gvl_elecylinder.fbi_gm_axisPickUp.out_flg_Done THEN
//				gvl_elecylinder.fbi_gm_axisTransport.in_flg_run := FALSE;
//				gvl_elecylinder.fbi_gm_axisPickUp.in_flg_run := FALSE;
//				var_process := 7;
//			END_IF
		7:
			gvl_io.flg_saftyUnitReset := FALSE;
			MC_ResetX.Execute := TRUE;
			MC_ResetY.Execute := TRUE;
			MC_ResetZ.Execute := TRUE;
			MC_ResetR.Execute := TRUE;
			gvl_elecylinder.ref_axis_transport.output.out_flg_reset := TRUE;
			gvl_elecylinder.ref_axis_sample.output.out_flg_reset := TRUE;
			gvl_elecylinder.ref_axis_trayChange.output.out_flg_reset := TRUE;
			gvl_elecylinder.ref_axis_rotary.output.out_flg_reset := TRUE;
			var_process := 8;
		8:
			MC_ResetX.Execute := FALSE;
			MC_ResetY.Execute := FALSE;
			MC_ResetZ.Execute := FALSE;
			MC_ResetR.Execute := FALSE;
			gvl_elecylinder.ref_axis_transport.output.out_flg_reset := FALSE;
			gvl_elecylinder.ref_axis_sample.output.out_flg_reset := FALSE;
			gvl_elecylinder.ref_axis_trayChange.output.out_flg_reset := FALSE;
			gvl_elecylinder.ref_axis_rotary.output.out_flg_reset := FALSE;
			fbi_delayTimer4.IN := TRUE;
			(*
			IF fbi_delayTimer4.Q THEN
				var_process := 6;
			END_IF
			*)
			IF gvl_io.in_wire_saftyUnitState THEN
				var_process := 9;
			ELSIF fbi_delayTimer4.Q THEN
				var_process := 9;
			END_IF
		9:	
			gvl_error.flg_resetEventFlg := TRUE;
			fbi_delayTimer1.IN := TRUE;
			IF fbi_delayTimer1.Q THEN
				var_process := 10;
			END_IF
		10:
			gvl_error.flg_eventDisplayRest := TRUE;
			fbi_delayTimer2.IN := TRUE;
			IF fbi_delayTimer2.Q THEN
				var_process := 11;
			END_IF
		11:
			fbi_delayTimer3.IN := TRUE;
			gvl_error.flg_ararmLevelRest := TRUE;
			IF fbi_delayTimer3.Q  THEN
				var_process := 12;
			END_IF
		12:
			gvl_error.flg_resetEventFlg := FALSE;
			gvl_error.flg_eventDisplayRest := FALSE;
			gvl_error.flg_ararmLevelRest := FALSE;
			gvl_error.flg_alramBusy := FALSE;
						
	END_CASE
END_IF
MC_ResetX(
	Axis:= gvl_axis.axisX , 
	Execute:= , 
	Done=> , 
	Busy=> , 
	Error=> , 
	ErrorID=> );
MC_ResetY(
	Axis:= gvl_axis.axisY , 
	Execute:= , 
	Done=> , 
	Busy=> , 
	Error=> , 
	ErrorID=> );
MC_ResetZ(
	Axis:= gvl_axis.axisZ , 
	Execute:= , 
	Done=> , 
	Busy=> , 
	Error=> , 
	ErrorID=> );
MC_ResetR(
	Axis:= gvl_axis.axisR , 
	Execute:= , 
	Done=> , 
	Busy=> , 
	Error=> , 
	ErrorID=> );
MC_Stop_x(
	Axis:= gvl_axis.axisX, 
	Execute:= , 
	Deceleration:= , 
	Jerk:= , 
	Options:= , 
	Done=> , 
	Busy=> , 
	Active=> , 
	CommandAborted=> , 
	Error=> , 
	ErrorID=> );
MC_Stop_y(
	Axis:= gvl_axis.axisY, 
	Execute:= , 
	Deceleration:= , 
	Jerk:= , 
	Options:= , 
	Done=> , 
	Busy=> , 
	Active=> , 
	CommandAborted=> , 
	Error=> , 
	ErrorID=> );
MC_Stop_z(
	Axis:= gvl_axis.axisZ, 
	Execute:= , 
	Deceleration:= , 
	Jerk:= , 
	Options:= , 
	Done=> , 
	Busy=> , 
	Active=> , 
	CommandAborted=> , 
	Error=> , 
	ErrorID=> );
MC_Stop_r(
	Axis:= gvl_axis.axisR, 
	Execute:= , 
	Deceleration:= , 
	Jerk:= , 
	Options:= , 
	Done=> , 
	Busy=> , 
	Active=> , 
	CommandAborted=> , 
	Error=> , 
	ErrorID=> );
	
	
fbi_delayTimer0(IN:= , PT:=T#500MS , Q=> , ET=> );
fbi_delayTimer1(IN:= , PT:=T#1000MS , Q=> , ET=> );
fbi_delayTimer2(IN:= , PT:=T#100MS , Q=> , ET=> );
fbi_delayTimer3(IN:= , PT:=T#100MS , Q=> , ET=> );
fbi_delayTimer4(IN:= , PT:=T#9000MS , Q=> , ET=> );
fbi_paramInit(in_flg_run:= , out_flg_done=> );
END_ACTION

ACTION manual_active:

IF manual._x AND manual.x = FALSE THEN
	gvl_io.flg_signalTowerGreen := FALSE;
	gvl_io.flg_signalTowerYellow := TRUE;
	gvl_io.flg_signalTowerRed := FALSE;
	gvl_visu.flg_btn_sample := FALSE;
	trn_autoRun := FALSE;
	gvl_visu.flg_btn_autoModeStart := FALSE;
	gvl_gm.var_incjetInfo.flg_denyStamp := FALSE;
	THIS^.fbi_manual();
	THIS^.fbi_manual.p_Init := TRUE;
ELSIF manual._x AND manual.x THEN
	THIS^.fbi_manual();
	THIS^.fbi_manual.p_Init := FALSE;
	gvl_auto.flg_transportClosed := FALSE;
	gvl_param.var_currentMode := eP_programMode.manual;
	gvl_io.flg_requestLens := FALSE;
	IF gvl_visu.flg_btn_autoModeStart THEN
		trn_autoRun := TRUE;
	END_IF
	gvl_param.var_productInfo[gvl_param.var_currentProductID].manaulVels.x.acc := 10000;
	gvl_param.var_productInfo[gvl_param.var_currentProductID].manaulVels.x.dcc := 10000;
	gvl_param.var_productInfo[gvl_param.var_currentProductID].manaulVels.y.acc := 10000;
	gvl_param.var_productInfo[gvl_param.var_currentProductID].manaulVels.y.dcc := 10000;
	gvl_param.var_productInfo[gvl_param.var_currentProductID].manaulVels.z.acc := 10000;
	gvl_param.var_productInfo[gvl_param.var_currentProductID].manaulVels.z.dcc := 10000;
 
	gvl_axis.ref_x.Velocity 	:= gvl_param.var_productInfo[gvl_param.var_currentProductID].manaulVels.x.vel;
	gvl_axis.ref_x.Acceleration := gvl_param.var_productInfo[gvl_param.var_currentProductID].manaulVels.x.acc;
	gvl_axis.ref_x.Deceleration := gvl_param.var_productInfo[gvl_param.var_currentProductID].manaulVels.x.dcc;
	gvl_axis.ref_y.Velocity 	:= gvl_param.var_productInfo[gvl_param.var_currentProductID].manaulVels.y.vel;
	gvl_axis.ref_y.Acceleration := gvl_param.var_productInfo[gvl_param.var_currentProductID].manaulVels.y.acc;
	gvl_axis.ref_y.Deceleration := gvl_param.var_productInfo[gvl_param.var_currentProductID].manaulVels.y.dcc;
	gvl_axis.ref_z.Velocity 	:= gvl_param.var_productInfo[gvl_param.var_currentProductID].manaulVels.z.vel;
	gvl_axis.ref_z.Acceleration := gvl_param.var_productInfo[gvl_param.var_currentProductID].manaulVels.z.acc;
	gvl_axis.ref_z.Deceleration := gvl_param.var_productInfo[gvl_param.var_currentProductID].manaulVels.z.dcc;
	gvl_axis.ref_r.Velocity 	:= gvl_gm.var_buf_manualVel;
END_IF
END_ACTION

PROPERTY p_init : bool
GET
p_init := THIS^.SFCInit;
END_GET
SET
THIS^.SFCInit := p_init;
END_SET
END_PROPERTY

ACTION SaftyUnitReset_active:
IF SaftyUnitReset._x AND SaftyUnitReset.x = FALSE THEN
	trn_SaftyUnitResetDone := FALSE;
	resetDelay.IN := FALSE;
	fbi_timer.IN := FALSE;
	gvl_io.flg_saftyUnitReset := TRUE;
	gvl_gm.var_incjetInfo.flg_denyStamp := FALSE;
ELSIF SaftyUnitReset._x AND SaftyUnitReset.x THEN
	resetDelay.IN := TRUE;
	fbi_timer.IN := True;
	IF resetDelay.Q THEN
		gvl_io.flg_saftyUnitReset := FALSE;
	END_IF
	
	IF gvl_io.flg_saftyUnitState THEN
		gvl_io.flg_saftyUnitReset := FALSE;
		trn_SaftyUnitResetDone := TRUE;
	ELSIF fbi_timer.Q THEN
		gvl_io.flg_saftyUnitReset := FALSE;
		trn_SaftyUnitResetDone := TRUE;
	END_IF
END_IF
resetDelay(IN:= , PT:=T#0.5S , Q=> , ET=> );
fbi_timer(IN:= , PT:=T#9S , Q=> , ET=> );
END_ACTION

END_FUNCTION_BLOCK

// ---- FBs/fb_manual.TcPOU
FUNCTION_BLOCK fb_manual
VAR_INPUT
END_VAR
VAR_OUTPUT
END_VAR
VAR
	SFCInit : BOOL;
	fbi_paramInit: fb_paramInit;
	trn_paramInitDone: BOOL;

	fbi_jogController: fb_jogController;
	fbi_PTP : fb_PTP;
	fbi_operationElecylinder : fb_operationElecylinder;
	fbi_gm_operationElecylinder :fb_gm_operationElecylinder;
	fbi_oeprationChuck : fb_oeprationChuck;
	fbi_oeprationPush :fb_oeprationPush;
	fbi_operationEjector : fb_operationEjector;
	fbi_gm_operationEjector : fb_gm_operationEjector;
	fbi_recordingSystem : fb_recordingSystem;
	fbi_productGenerater : fb_productGenerator;
	fbi_gm_operationSV	: fb_gm_operationSV;
	var_i: INT;
	fbi_gm_setting: fb_gm_setting;
	fbi_gm_PTP: fb_gm_PTP;
	fbi_debugData: fb_debugData;
	var_cav_i: INT;
END_VAR

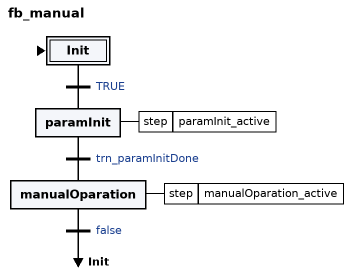
INITIAL_STEP Init:
END_STEP
TRANSITION FROM Init TO paramInit
    := TRUE;
END_TRANSITION
STEP paramInit:
    paramInit_active(N);  // step action
END_STEP
TRANSITION FROM paramInit TO manualOparation
    := trn_paramInitDone;
END_TRANSITION
STEP manualOparation:
    manualOparation_active(N);  // step action
END_STEP
TRANSITION FROM manualOparation TO Init
    := false;
END_TRANSITION

ACTION manualOparation_active:
IF manualOparation._x AND manualOparation.x = FALSE THEN
	THIS^.fbi_PTP();
	THIS^.fbi_PTP.p_init := TRUE;
	THIS^.fbi_operationElecylinder();
	THIS^.fbi_operationElecylinder.p_Init := TRUE;
	THIS^.fbi_gm_operationElecylinder();
	THIS^.fbi_gm_operationElecylinder.p_Init := TRUE;
	THIS^.fbi_oeprationChuck();
	THIS^.fbi_oeprationChuck.p_Init := TRUE;
	THIS^.fbi_oeprationPush();
	THIS^.fbi_oeprationPush.p_Init := TRUE;
	THIS^.fbi_operationEjector();
	THIS^.fbi_operationEjector.p_Init := TRUE;
	THIS^.fbi_gm_operationEjector();
	THIS^.fbi_gm_operationEjector.p_Init := TRUE;
	THIS^.fbi_gm_operationSV();
	THIS^.fbi_gm_operationSV.p_Init := TRUE;
	fbi_gm_PTP(in_flg_run := FALSE);
	//test mode
	fbi_debugData();
ELSIF manualOparation._x AND manualOparation.x THEN
	
//operation jog
	THIS^.fbi_jogController();
//PTP
	THIS^.fbi_PTP();
	THIS^.fbi_PTP.p_init := FALSE;
	fbi_gm_PTP(in_flg_run := TRUE);
//operation elecylinder
	THIS^.fbi_operationElecylinder();
	THIS^.fbi_operationElecylinder.p_Init := FALSE;
	THIS^.fbi_gm_operationElecylinder();
	THIS^.fbi_gm_operationElecylinder.p_Init := FALSE;
//operation chuck
	THIS^.fbi_oeprationChuck();
	THIS^.fbi_oeprationChuck.p_Init := FALSE;
	THIS^.fbi_gm_operationSV();
	THIS^.fbi_gm_operationSV.p_Init := FALSE;
//operation push
	THIS^.fbi_oeprationPush();
	THIS^.fbi_oeprationPush.p_Init := FALSE;
//operation ejector
	THIS^.fbi_operationEjector();
	THIS^.fbi_operationEjector.p_Init := FALSE;
	THIS^.fbi_gm_operationEjector();
	THIS^.fbi_gm_operationEjector.p_Init := FALSE;
//recording teach position
	THIS^.fbi_recordingSystem();
	fbi_gm_setting();
//new product generater
	THIS^.fbi_productGenerater();
//reset defective qty
	IF gvl_visu.flg_btn_clrDefectiveQty THEN
		FOR var_i := 1 TO 8 BY 1 DO
			gvl_auto.var_defectiveLens[var_i] := 0;
		END_FOR
	END_IF
//reset pocket qty
	IF gvl_visu.flg_btn_clrPockertQty THEN
		gvl_auto.flg_pocketCountCheck := false;
		FOR var_i := 1 TO 8 BY 1 DO
			gvl_auto.pocketNo[var_i] := 0;
		END_FOR
	END_IF
//reset gate length data
	IF gvl_visu.flg_btn_clrGateData THEN
		FOR var_i := 49 TO 0 BY -1 DO
			gvl_visu.var_gateLengthList[var_i] := 0;
			FOR var_cav_i := 1 TO 8 DO
				gvl_visu.var_gateLengthListCav[var_cav_i][var_i] := 0;
			END_FOR
		END_FOR
	END_IF
END_IF
//gate measurement run preset
	IF gvl_visu.flg_btn_gateMeasurementPreset THEN
		gvl_io.var_gateMeasurementPreset := 1;
	ELSE
		gvl_io.var_gateMeasurementPreset := 0;
	END_IF
END_ACTION

PROPERTY p_Init : bool
GET
p_init := THIS^.SFCInit;
END_GET
SET
THIS^.SFCInit := p_init;
END_SET
END_PROPERTY

ACTION paramInit_active:
fbi_paramInit(in_flg_run:= , out_flg_done=> );
IF paramInit._x AND paramInit.x = FALSE THEN
	trn_paramInitDone:= FALSE;
	fbi_paramInit.in_flg_run := FALSE;
ELSIF paramInit._x AND paramInit.x THEN
	fbi_paramInit.in_flg_run := TRUE;
	IF fbi_paramInit.out_flg_done THEN
		fbi_paramInit.in_flg_run := FALSE;
		trn_paramInitDone := TRUE;
	END_IF
END_IF
END_ACTION

END_FUNCTION_BLOCK

// ---- FBs/fb_paramInit.TcPOU
FUNCTION_BLOCK fb_paramInit
VAR_INPUT
	in_flg_run : BOOL;
END_VAR
VAR_OUTPUT
	out_flg_done : BOOL;
END_VAR
VAR
	flg_busy: bool;
	fbi_eje_reset: fb_eje_reset;
	fbi_r_TRIG: R_TRIG;
	fbi_sv_reset: fb_sv_reset;
	fbi_sv_pushReset: fb_sv_reset;
	fbi_ele_reset: ARRAY[1..6] OF fb_ele_reset;
	fbi_ton1: TON;
	fbi_ton2: TON;
	var_process: INT;
	fbi_gm_eje_reset : fb_eje_reset;
	fbi_gm_sv_reset: fb_sv_reset;
	fbi_gm_sv_pushReset: fb_sv_reset;
	fbi_gm_sv_rotaryReset: fb_sv_reset;
	fbi_gm_sv_pickUpReset: fb_sv_reset;
	fbi_gm_sv_stampReset: fb_sv_reset;
END_VAR

fbi_r_TRIG(CLK:= in_flg_run, Q=> );
IF fbi_r_TRIG.Q THEN
	
	var_process := 0;
	flg_busy := TRUE;
END_IF
IF NOT in_flg_run THEN
	fbi_ton1.in := FALSE;
	fbi_ton2.IN := FALSE;
	var_process := 0;
	out_flg_done := FALSE;
	flg_busy := FALSE;
END_IF
//motor
CASE var_process OF
	0:
		gvl_visu.flg_powerOn := FALSE;
		gvl_axis.ref_x.Execute := FALSE;
		gvl_axis.ref_y.Execute := FALSE;
		gvl_axis.ref_z.Execute := FALSE;
		gvl_axis.ref_r.Execute := FALSE;
		
		gvl_axis.fbi_mc_jogX.JogForward := FALSE;
		gvl_axis.fbi_mc_jogX.JogBackwards := FALSE;
		gvl_axis.fbi_mc_jogY.JogForward := FALSE;
		gvl_axis.fbi_mc_jogY.JogBackwards := FALSE;
		gvl_axis.fbi_mc_jogZ.JogForward := FALSE;
		gvl_axis.fbi_mc_jogZ.JogBackwards := FALSE;
		gvl_axis.fbi_mc_jogR.JogForward := FALSE;
		gvl_axis.fbi_mc_jogR.JogBackwards := FALSE;
		
		gvl_axis.fbi_motionControler.in_flg_start := FALSE;
		
		//elecylinder , solv
		gvl_solv.fbi_ejector.in_flg_run := FALSE;
		gvl_solv.fbi_chuck.in_flg_run := FALSE;
		gvl_solv.fbi_push.in_flg_run := FALSE;
		
		
		gvl_solv.fbi_gm_ejector.in_flg_run := FALSE;
		gvl_solv.fbi_gm_chuck.in_flg_run := FALSE;
		gvl_solv.fbi_gm_push.in_flg_run := FALSE;
		gvl_solv.fbi_gm_rotary.in_flg_run := FALSE;
		gvl_solv.fbi_gm_pickup.in_flg_run := FALSE;
		gvl_solv.fbi_gm_stamp.in_flg_run := FALSE;
		
		gvl_elecylinder.fbi_axisTransport.in_flg_run := FALSE;
		gvl_elecylinder.fbi_axisSample.in_flg_run := FALSE;
		gvl_elecylinder.fbi_axisTrayChange.in_flg_run := FALSE;
		gvl_elecylinder.fbi_axisRotary.in_flg_run := FALSE;
		gvl_elecylinder.fbi_gm_axisPickUp.in_flg_run := FALSE;
		gvl_elecylinder.fbi_gm_axisTransport.in_flg_run := FALSE;
		fbi_ton2.IN := TRUE;
		
		gvl_solv.fbi_ejector.in_var_vacMode := eP_ejeVacMode.halt;
		gvl_solv.fbi_chuck.in_var_moveMode := eP_svMovemode.stop;
		gvl_solv.fbi_push.in_var_moveMode := eP_svMovemode.stop;
		
		gvl_solv.fbi_gm_ejector.in_var_vacMode := eP_ejeVacMode.halt;
		gvl_solv.fbi_gm_chuck.in_var_moveMode := eP_svMovemode.stop;
		gvl_solv.fbi_gm_push.in_var_moveMode := eP_svMovemode.stop;
		gvl_solv.fbi_gm_rotary.in_var_moveMode := eP_svMovemode.stop;
		gvl_solv.fbi_gm_pickup.in_var_moveMode := eP_svMovemode.stop;
		gvl_solv.fbi_gm_stamp.in_var_moveMode := eP_svMovemode.stop;
		
		
		gvl_elecylinder.fbi_axisTransport.in_var_moveMode := eP_eleMovemode.stop;
		gvl_elecylinder.fbi_axisSample.in_var_moveMode := eP_eleMovemode.stop;
		gvl_elecylinder.fbi_axisTrayChange.in_var_moveMode := eP_eleMovemode.stop;
		gvl_elecylinder.fbi_axisRotary.in_var_moveMode := eP_eleMovemode.stop;
		gvl_elecylinder.fbi_gm_axisPickUp.in_var_moveMode := eP_eleMovemode.stop;
		gvl_elecylinder.fbi_gm_axisTransport.in_var_moveMode := eP_eleMovemode.stop;
		
		gvl_io.flg_requestLens := FALSE;

		
		IF fbi_ton2.Q THEN
			var_process := 1;
		END_IF
	1:
	
		gvl_axis.fbi_motionControler.p_Init := FALSE;
		var_process := 2;

	2:
		flg_busy := FALSE;
		fbi_ton1.IN := TRUE;
		out_flg_done := TRUE;
		var_process := 3;
	3:
		out_flg_done := FALSE;
END_CASE
fbi_ton1(IN:= , PT:=T#500MS , Q=> , ET=> );
fbi_ton2(IN:= , PT:=T#500MS , Q=> , ET=> );
fbi_eje_reset(var_ref_eje:=gvl_solv.ref_ejector , in_flg_reset:=flg_busy , out_flg_resetDone=> );
fbi_sv_reset(var_ref_sv:= gvl_solv.ref_chuck, in_flg_reset:= flg_busy, out_flg_resetDone=> );
fbi_sv_pushReset(var_ref_sv:= gvl_solv.ref_push, in_flg_reset:= flg_busy, out_flg_resetDone=> );
fbi_gm_eje_reset(var_ref_eje:=gvl_solv.ref_gm_ejctor, in_flg_reset:=flg_busy , out_flg_resetDone=> );
fbi_gm_sv_reset(var_ref_sv:= gvl_solv.ref_gm_chuck, in_flg_reset:= flg_busy, out_flg_resetDone=> );
fbi_gm_sv_pushReset(var_ref_sv:= gvl_solv.ref_gm_push, in_flg_reset:= flg_busy, out_flg_resetDone=> );
fbi_gm_sv_rotaryReset(var_ref_sv:= gvl_solv.ref_gm_rotary, in_flg_reset:= flg_busy, out_flg_resetDone=> );
fbi_gm_sv_pickUpReset(var_ref_sv:= gvl_solv.ref_gm_pickUp, in_flg_reset:= flg_busy, out_flg_resetDone=> );
fbi_gm_sv_stampReset(var_ref_sv:= gvl_solv.ref_gm_stamp, in_flg_reset:= flg_busy, out_flg_resetDone=> );
fbi_ele_reset[1](var_ref_ele:= gvl_elecylinder.ref_axis_transport, in_flg_reset:= flg_busy, out_flg_resetDone=> );
fbi_ele_reset[2](var_ref_ele:= gvl_elecylinder.ref_axis_sample, in_flg_reset:= flg_busy, out_flg_resetDone=> );
fbi_ele_reset[3](var_ref_ele:= gvl_elecylinder.ref_axis_trayChange, in_flg_reset:= flg_busy, out_flg_resetDone=> );
fbi_ele_reset[4](var_ref_ele:= gvl_elecylinder.ref_axis_rotary, in_flg_reset:= flg_busy, out_flg_resetDone=> );
fbi_ele_reset[5](var_ref_ele:= gvl_elecylinder.ref_gm_axisPickUp, in_flg_reset:= flg_busy, out_flg_resetDone=> );
fbi_ele_reset[6](var_ref_ele:= gvl_elecylinder.ref_gm_axisTransport, in_flg_reset:= flg_busy, out_flg_resetDone=> );

END_FUNCTION_BLOCK

// ---- FBs/fb_ejecter/fb_eje_reset.TcPOU
FUNCTION_BLOCK fb_eje_reset
VAR_IN_OUT
	var_ref_eje : ref_eje_io;
END_VAR
VAR_INPUT
	in_flg_reset : BOOL;
END_VAR
VAR_OUTPUT
	out_flg_resetDone: BOOL;
END_VAR
VAR

	fbi_ton1: TON;
	var_process: INT;
END_VAR


fbi_ton1(IN:= , PT:=T#100MS , Q=> , ET=> );

IF NOT in_flg_reset THEN
	var_process := 0;
END_IF
CASE var_process OF
	0:
		IF in_flg_reset THEN
			var_process := 1;
		END_IF
	1:
		fbi_ton1.IN := FALSE;
		var_process := 2;
	2:	
		fbi_ton1.IN := TRUE;
		var_ref_eje.param.var_mutex := 0;
		var_ref_eje.output.out_flg_ejeVac := FALSE;
		var_ref_eje.output.out_flg_ejeBrk := FALSE;
		IF fbi_ton1.Q THEN
			var_process := 3;
		END_IF
	3:
		out_flg_resetDone := TRUE;
		var_process := 4;
	4:
		out_flg_resetDone := FALSE;
END_CASE

END_FUNCTION_BLOCK

// ---- FBs/fb_sv/fb_sv_reset.TcPOU
FUNCTION_BLOCK fb_sv_reset
VAR_IN_OUT
	var_ref_sv : ref_sv_io;
END_VAR
VAR_INPUT
	in_flg_reset : BOOL;
END_VAR
VAR_OUTPUT
	out_flg_resetDone: BOOL;
END_VAR
VAR

	var_process: INT;
	fbi_ton1: TON;
END_VAR


fbi_ton1(IN:= , PT:=T#100MS , Q=> , ET=> );

IF NOT in_flg_reset THEN
	var_process := 0;
END_IF
CASE var_process OF
	0:
		IF in_flg_reset THEN
			fbi_ton1.IN := FALSE;
			var_process := 1;
		END_IF
	1:	
		fbi_ton1.IN := TRUE;
		var_ref_sv.out.out_flg_svA := FALSE;
		var_ref_sv.out.out_flg_svB := FALSE;
		var_ref_sv.param.var_mutex := 0;
		IF fbi_ton1.Q THEN
			var_process := 2;
		END_IF
	2:
		out_flg_resetDone := TRUE;
		var_process := 3;
	3:
		out_flg_resetDone := FALSE;
END_CASE

END_FUNCTION_BLOCK

// ---- FBs/fb_ele/fb_ele_reset.TcPOU
FUNCTION_BLOCK fb_ele_reset
VAR_IN_OUT
	var_ref_ele : ref_ele_io;
END_VAR
VAR_INPUT
	in_flg_reset : BOOL;
END_VAR
VAR_OUTPUT
	out_flg_resetDone : bool;
END_VAR
VAR
	var_process: INT;
	fbi_ton1: TON;
END_VAR


fbi_ton1(IN:= , PT:=T#100MS , Q=> , ET=> );
IF NOT in_flg_reset THEN
	var_process := 0;
	out_flg_resetDone := FALSE;
	var_ref_ele.output.out_flg_reset := FALSE;
END_IF
CASE var_process OF
	0:
		IF in_flg_reset THEN
			fbi_ton1.IN := FALSE;
			var_process := 1;
		END_IF
	1:
		var_ref_ele.output.out_flg_eleA := FALSE;
		var_ref_ele.output.out_flg_eleB := FALSE;
		var_ref_ele.output.out_flg_reset := TRUE;
		var_ref_ele.param.var_mutex := 0;
		fbi_ton1.IN := TRUE;
		IF fbi_ton1.Q THEN
			var_process := 2;
		END_IF
	2:
		var_ref_ele.output.out_flg_reset := FALSE;
		out_flg_resetDone := TRUE;
		var_process := 3;
	3:
		out_flg_resetDone := FALSE;
END_CASE

END_FUNCTION_BLOCK

// ---- FBs/fb_jogController.TcPOU
FUNCTION_BLOCK fb_jogController
VAR_INPUT
END_VAR
VAR_OUTPUT
END_VAR
VAR
END_VAR

CASE gvl_visu.var_jofAxis OF
		eP_xyz.x:
			IF gvl_visu.flg_btn_moveDirct = eP_direction.positive OR gvl_io.flg_btnGreen THEN
				gvl_axis.fbi_mc_jogX.JogForward := TRUE;
				gvl_axis.fbi_mc_jogX.JogBackwards := FALSE;
			ELSIF gvl_visu.flg_btn_moveDirct = eP_direction.negative OR gvl_io.flg_btnRed THEN
				gvl_axis.fbi_mc_jogX.JogForward := FALSE;
				gvl_axis.fbi_mc_jogX.JogBackwards := TRUE;
			ELSE
				gvl_axis.fbi_mc_jogX.JogForward := FALSE;
				gvl_axis.fbi_mc_jogX.JogBackwards := FALSE;
			END_IF
		eP_xyz.y:
			IF gvl_visu.flg_btn_moveDirct = eP_direction.positive OR gvl_io.flg_btnGreen THEN
				gvl_axis.fbi_mc_jogY.JogForward := TRUE;
				gvl_axis.fbi_mc_jogY.JogBackwards := FALSE;
			ELSIF gvl_visu.flg_btn_moveDirct = eP_direction.negative OR gvl_io.flg_btnRed THEN
				gvl_axis.fbi_mc_jogY.JogForward := FALSE;
				gvl_axis.fbi_mc_jogY.JogBackwards := TRUE;
			ELSE
				gvl_axis.fbi_mc_jogY.JogForward := FALSE;
				gvl_axis.fbi_mc_jogY.JogBackwards := FALSE;
			END_IF
		eP_xyz.z:
			IF gvl_visu.flg_btn_moveDirct = eP_direction.positive OR gvl_io.flg_btnGreen THEN
				gvl_axis.fbi_mc_jogZ.JogForward := TRUE;
				gvl_axis.fbi_mc_jogZ.JogBackwards := FALSE;
			ELSIF gvl_visu.flg_btn_moveDirct = eP_direction.negative OR gvl_io.flg_btnRed THEN
				gvl_axis.fbi_mc_jogZ.JogForward := FALSE;
				gvl_axis.fbi_mc_jogZ.JogBackwards := TRUE;
			ELSE
				gvl_axis.fbi_mc_jogZ.JogForward := FALSE;
				gvl_axis.fbi_mc_jogZ.JogBackwards := FALSE;
			END_IF
END_CASE
CASE gvl_visu.var_radio_jogMode OF
	0:
		gvl_axis.fbi_mc_jogX.Mode := E_JogMode.MC_JOGMODE_INCHING;
		gvl_axis.fbi_mc_jogY.Mode := E_JogMode.MC_JOGMODE_INCHING;
		gvl_axis.fbi_mc_jogZ.Mode := E_JogMode.MC_JOGMODE_INCHING;
	1:
		gvl_axis.fbi_mc_jogX.Mode := E_JogMode.MC_JOGMODE_CONTINOUS;
		gvl_axis.fbi_mc_jogY.Mode := E_JogMode.MC_JOGMODE_CONTINOUS;
		gvl_axis.fbi_mc_jogZ.Mode := E_JogMode.MC_JOGMODE_CONTINOUS;
END_CASE
gvl_axis.fbi_mc_jogX.Position := gvl_visu.var_in_inch;
gvl_axis.fbi_mc_jogY.Position := gvl_visu.var_in_inch;
gvl_axis.fbi_mc_jogZ.Position := gvl_visu.var_in_inch;

END_FUNCTION_BLOCK

// ---- FBs/fb_PTP.TcPOU
FUNCTION_BLOCK fb_PTP
VAR_INPUT
END_VAR
VAR_OUTPUT
END_VAR
VAR
	SFCInit : BOOL;
	trn_PosInitDone: BOOL;
	trn_PosPickUpDone: BOOL;
	trn_PosRemoveDone: BOOL;
	trn_PosSampleDone: BOOL;
	trn_PosPocketDone: BOOL;
	fbi_R_TRIG: ARRAY [0..6] OF R_TRIG;
	flg_moveRun: BOOL;
	flg_moveDone: BOOL;
	trn_caluculateDone: BOOL;
	fbi_coordinateCal: fb_coordinateCal;
	fbi_CycleDelayTimer: ARRAY[0..6] OF TON;
	fbi_axisZ_R_TRIG:ARRAY[0..6] OF R_TRIG;
	trn_Mode1Done: BOOL;
	trn_Mode2Done: BOOL;
	var_targetPosX: LREAL;
	var_targetPosY: LREAL;
	var_targetPosZ: LREAL;
	trn_PassPosDone: BOOL;
	trn_SetPosDone: BOOL;
	var_process: INT;
	trn_move_all_done: BOOL;
	var_in_all_pocketNo: INT;
	flg_stop: BOOL;
END_VAR

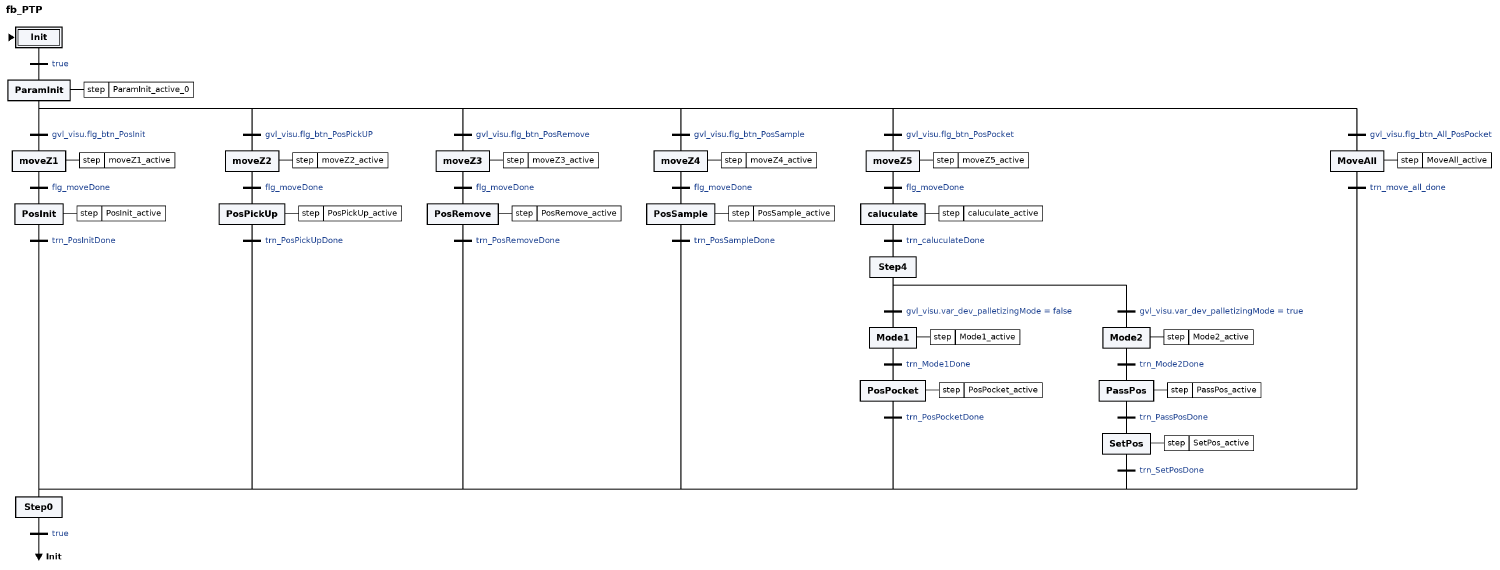
INITIAL_STEP Init:
END_STEP
TRANSITION FROM Init TO ParamInit
    := true;
END_TRANSITION
STEP ParamInit:
    ParamInit_active_0(N);  // step action
END_STEP
TRANSITION FROM ParamInit TO moveZ1
    := gvl_visu.flg_btn_PosInit;
END_TRANSITION
STEP moveZ1:
    moveZ1_active(N);  // step action
END_STEP
TRANSITION FROM moveZ1 TO PosInit
    := flg_moveDone;
END_TRANSITION
STEP PosInit:
    PosInit_active(N);  // step action
END_STEP
TRANSITION FROM PosInit TO Step0
    := trn_PosInitDone;
END_TRANSITION
TRANSITION FROM ParamInit TO moveZ2
    := gvl_visu.flg_btn_PosPickUP;
END_TRANSITION
STEP moveZ2:
    moveZ2_active(N);  // step action
END_STEP
TRANSITION FROM moveZ2 TO PosPickUp
    := flg_moveDone;
END_TRANSITION
STEP PosPickUp:
    PosPickUp_active(N);  // step action
END_STEP
TRANSITION FROM PosPickUp TO Step0
    := trn_PosPickUpDone;
END_TRANSITION
TRANSITION FROM ParamInit TO moveZ3
    := gvl_visu.flg_btn_PosRemove;
END_TRANSITION
STEP moveZ3:
    moveZ3_active(N);  // step action
END_STEP
TRANSITION FROM moveZ3 TO PosRemove
    := flg_moveDone;
END_TRANSITION
STEP PosRemove:
    PosRemove_active(N);  // step action
END_STEP
TRANSITION FROM PosRemove TO Step0
    := trn_PosRemoveDone;
END_TRANSITION
TRANSITION FROM ParamInit TO moveZ4
    := gvl_visu.flg_btn_PosSample;
END_TRANSITION
STEP moveZ4:
    moveZ4_active(N);  // step action
END_STEP
TRANSITION FROM moveZ4 TO PosSample
    := flg_moveDone;
END_TRANSITION
STEP PosSample:
    PosSample_active(N);  // step action
END_STEP
TRANSITION FROM PosSample TO Step0
    := trn_PosSampleDone;
END_TRANSITION
TRANSITION FROM ParamInit TO moveZ5
    := gvl_visu.flg_btn_PosPocket;
END_TRANSITION
STEP moveZ5:
    moveZ5_active(N);  // step action
END_STEP
TRANSITION FROM moveZ5 TO caluculate
    := flg_moveDone;
END_TRANSITION
STEP caluculate:
    caluculate_active(N);  // step action
END_STEP
TRANSITION FROM caluculate TO Step4
    := trn_caluculateDone;
END_TRANSITION
STEP Step4:
END_STEP
TRANSITION FROM Step4 TO Mode1
    := gvl_visu.var_dev_palletizingMode = false;
END_TRANSITION
STEP Mode1:
    Mode1_active(N);  // step action
END_STEP
TRANSITION FROM Mode1 TO PosPocket
    := trn_Mode1Done;
END_TRANSITION
STEP PosPocket:
    PosPocket_active(N);  // step action
END_STEP
TRANSITION FROM PosPocket TO Step0
    := trn_PosPocketDone;
END_TRANSITION
TRANSITION FROM Step4 TO Mode2
    := gvl_visu.var_dev_palletizingMode = true;
END_TRANSITION
STEP Mode2:
    Mode2_active(N);  // step action
END_STEP
TRANSITION FROM Mode2 TO PassPos
    := trn_Mode2Done;
END_TRANSITION
STEP PassPos:
    PassPos_active(N);  // step action
END_STEP
TRANSITION FROM PassPos TO SetPos
    := trn_PassPosDone;
END_TRANSITION
STEP SetPos:
    SetPos_active(N);  // step action
END_STEP
TRANSITION FROM SetPos TO Step0
    := trn_SetPosDone;
END_TRANSITION
TRANSITION FROM ParamInit TO MoveAll
    := gvl_visu.flg_btn_All_PosPocket;
END_TRANSITION
STEP MoveAll:
    MoveAll_active(N);  // step action
END_STEP
TRANSITION FROM MoveAll TO Step0
    := trn_move_all_done;
END_TRANSITION
STEP Step0:
END_STEP
TRANSITION FROM Step0 TO Init
    := true;
END_TRANSITION

ACTION caluculate_active:
IF caluculate._x AND caluculate.x = FALSE THEN
	trn_caluculateDone:= FALSE;
	fbi_coordinateCal.in_flg_run := FALSE;
ELSIF caluculate._x AND caluculate.x THEN
	fbi_coordinateCal.in_flg_run := TRUE;
	IF fbi_coordinateCal.out_flg_Done THEN
		trn_caluculateDone := TRUE;
	END_IF
END_IF

fbi_coordinateCal(
	in_flg_run:= , 
	out_flg_run=> , 
	var_ref_productInfo:= gvl_param.var_productInfo[gvl_param.var_currentProductID], 
	in_var_cavNo:= gvl_visu.var_in_cavNo, 
	in_var_pocketNo:= gvl_visu.var_in_pocketNo, 
	in_var_calculateMode:= , 
	out_flg_busy=> , 
	out_flg_Done=> , 
	out_var_X=> var_targetPosX, 
	out_var_Y=> var_targetPosY, 
	out_var_Z=> var_targetPosZ
);
END_ACTION

ACTION Mode1_active:
IF Mode1._x AND Mode1.x = FALSE THEN
	trn_Mode1Done := FALSE;
	gvl_axis.fbi_motionControler.in_var_targetPosX := var_targetPosX;
	gvl_axis.fbi_motionControler.in_var_targetPosY := var_targetPosY;
	gvl_axis.fbi_motionControler.in_var_targetPosZ := var_targetPosZ;
ELSIF Mode1._x AND Mode1.x THEN
	trn_Mode1Done := TRUE;
END_IF
END_ACTION

ACTION Mode2_active:
IF Mode2._x AND Mode2.x = FALSE THEN
	trn_Mode2Done := FALSE;
	gvl_axis.fbi_motionControler.in_var_targetPosX := var_targetPosX + gvl_param.var_productInfo[gvl_param.var_currentProductID].teachPos.palletize.upperLower[gvl_param.var_currentTrayPos].cav[gvl_visu.var_in_cavNo].teachingDetail.passingPos.x;
	gvl_axis.fbi_motionControler.in_var_targetPosY := var_targetPosY + gvl_param.var_productInfo[gvl_param.var_currentProductID].teachPos.palletize.upperLower[gvl_param.var_currentTrayPos].cav[gvl_visu.var_in_cavNo].teachingDetail.passingPos.y;
	gvl_axis.fbi_motionControler.in_var_targetPosZ := var_targetPosZ + gvl_param.var_productInfo[gvl_param.var_currentProductID].teachPos.palletize.upperLower[gvl_param.var_currentTrayPos].cav[gvl_visu.var_in_cavNo].teachingDetail.passingPos.z;
ELSIF Mode2._x AND Mode2.x THEN
	trn_Mode2Done := TRUE;
END_IF
END_ACTION

ACTION MoveAll_active:
IF MoveAll._x AND MoveAll.x = FALSE THEN
	var_process := 0;
	var_in_all_pocketNo:= 0;
	trn_move_all_done := FALSE;
	gvl_axis.ref_z.Execute := FALSE;
	fbi_coordinateCal.in_flg_run := FALSE;
	gvl_axis.fbi_motionControler.in_flg_start := FALSE;
	flg_stop:= FALSE;
	gvl_visu.flg_All_PosPorket_Move:= FALSE;
ELSIF MoveAll._x AND MoveAll.x THEN
	IF gvl_visu.flg_btn_autoModeStop THEN
		flg_stop:= TRUE;
	END_IF
	CASE var_process OF
		0:
			gvl_axis.ref_z.Position := 50;
			gvl_axis.ref_z.Execute := TRUE;
			fbi_CycleDelayTimer[6].IN := FALSE;
			var_in_all_pocketNo:= var_in_all_pocketNo + 1;
			var_process := 1;
		1:
			gvl_visu.flg_All_PosPorket_Move:= TRUE;
			IF gvl_axis.ref_z.Done THEN
				gvl_axis.ref_z.Execute := FALSE;
				var_process := 2;
			END_IF
		2:
			IF flg_stop THEN
				var_process := 8;
			ELSE
				fbi_coordinateCal.in_flg_run := TRUE;
				gvl_axis.fbi_motionControler.p_Init := TRUE;
				gvl_axis.fbi_motionControler.in_flg_start := FALSE;
				IF fbi_coordinateCal.out_flg_Done THEN
					fbi_coordinateCal.in_flg_run := FALSE;
					var_process := 3;
				END_IF
			END_IF
		3:
			gvl_visu.var_in_pocketNo := var_in_all_pocketNo;
			gvl_axis.fbi_motionControler.p_Init := FALSE;
			gvl_axis.fbi_motionControler.in_var_targetPosX := var_targetPosX;
			gvl_axis.fbi_motionControler.in_var_targetPosY := var_targetPosY;
			gvl_axis.fbi_motionControler.in_var_targetPosZ := var_targetPosZ;
			gvl_axis.fbi_motionControler.in_var_direction := eP_motionDirection.XYZ;
			gvl_axis.fbi_motionControler.in_flg_start := TRUE;
			var_process := 4;
		4:
			IF gvl_axis.fbi_motionControler.out_flg_Done THEN
				gvl_axis.fbi_motionControler.in_flg_start := FALSE;
				var_process := 5;
			END_IF
		5:
			fbi_CycleDelayTimer[6].IN := TRUE;
			var_process := 6;
		6:
			IF fbi_CycleDelayTimer[6].Q THEN
				fbi_CycleDelayTimer[6].IN := FALSE;
				var_process := 7;
			END_IF
		7:
			IF(var_in_all_pocketNo >= gvl_param.var_productInfo[gvl_param.var_currentProductID].pocketSumQty) THEN
				var_process := 8;
			ELSE
				var_process := 0;
			END_IF
		8:	
			gvl_visu.flg_All_PosPorket_Move:= FALSE;
			trn_move_all_done := TRUE;
			
	END_CASE
END_IF
fbi_CycleDelayTimer[6](IN:= , PT:=T#3000MS , Q=> , ET=> );
fbi_coordinateCal(
	in_flg_run:= , 
	out_flg_run=> , 
	var_ref_productInfo:= gvl_param.var_productInfo[gvl_param.var_currentProductID], 
	in_var_cavNo:= gvl_visu.var_in_cavNo, 
	in_var_pocketNo:= var_in_all_pocketNo, 
	in_var_calculateMode:= , 
	out_flg_busy=> , 
	out_flg_Done=> , 
	out_var_X=> var_targetPosX, 
	out_var_Y=> var_targetPosY, 
	out_var_Z=> var_targetPosZ
);
END_ACTION

ACTION moveZ1_active:
IF moveZ1._x AND moveZ1.x = FALSE THEN
	flg_moveDone := FALSE;
	gvl_axis.ref_z.Execute := FALSE;
	gvl_axis.ref_z.Position := 5;
	fbi_axisZ_R_TRIG[0].CLK := FALSE;
ELSIF moveZ1._x AND moveZ1.x THEN
	fbi_axisZ_R_TRIG[0].CLK := TRUE;
	IF gvl_axis.ref_z.Done THEN
		flg_moveDone := TRUE;
	END_IF
END_IF
fbi_axisZ_R_TRIG[0](CLK:= , Q=>gvl_axis.ref_z.Execute );
END_ACTION

ACTION moveZ2_active:
IF moveZ2._x AND moveZ2.x = FALSE THEN
	flg_moveDone := FALSE;
	gvl_axis.ref_z.Execute := FALSE;
	gvl_axis.ref_z.Position := 5;
	fbi_axisZ_R_TRIG[1].CLK := FALSE;
ELSIF moveZ2._x AND moveZ2.x THEN
	fbi_axisZ_R_TRIG[1].CLK := TRUE;
	IF gvl_axis.ref_z.Done THEN
		flg_moveDone := TRUE;
	END_IF
END_IF
fbi_axisZ_R_TRIG[1](CLK:= , Q=>gvl_axis.ref_z.Execute );
END_ACTION

ACTION moveZ3_active:
IF moveZ3._x AND moveZ3.x = FALSE THEN
	flg_moveDone := FALSE;
	gvl_axis.ref_z.Execute := FALSE;
	gvl_axis.ref_z.Position := 5;
	fbi_axisZ_R_TRIG[2].CLK := FALSE;
ELSIF moveZ3._x AND moveZ3.x THEN
	fbi_axisZ_R_TRIG[2].CLK := TRUE;
	IF gvl_axis.ref_z.Done THEN
		flg_moveDone := TRUE;
	END_IF
END_IF
fbi_axisZ_R_TRIG[2](CLK:= , Q=>gvl_axis.ref_z.Execute );
END_ACTION

ACTION moveZ4_active:
IF moveZ4._x AND moveZ4.x = FALSE THEN
	flg_moveDone := FALSE;
	gvl_axis.ref_z.Execute := FALSE;
	gvl_axis.ref_z.Position := 5;
	fbi_axisZ_R_TRIG[3].CLK := FALSE;
ELSIF moveZ4._x AND moveZ4.x THEN
	fbi_axisZ_R_TRIG[3].CLK := TRUE;
	IF gvl_axis.ref_z.Done THEN
		flg_moveDone := TRUE;
	END_IF
END_IF
fbi_axisZ_R_TRIG[3](CLK:= , Q=>gvl_axis.ref_z.Execute );
END_ACTION

ACTION moveZ5_active:
IF moveZ5._x AND moveZ5.x = FALSE THEN
	flg_moveDone := FALSE;
	gvl_axis.ref_z.Execute := FALSE;
	gvl_axis.ref_z.Position := 5;
	fbi_axisZ_R_TRIG[4].CLK := FALSE;
ELSIF moveZ5._x AND moveZ5.x THEN
	fbi_axisZ_R_TRIG[4].CLK := TRUE;
	IF gvl_axis.ref_z.Done THEN
		flg_moveDone := TRUE;
	END_IF
END_IF
fbi_axisZ_R_TRIG[4](CLK:= , Q=>gvl_axis.ref_z.Execute );
END_ACTION

PROPERTY p_init : bool
GET
p_init := THIS^.SFCInit;
END_GET
SET
THIS^.SFCInit := p_init;
END_SET
END_PROPERTY

ACTION ParamInit_active_0:

IF ParamInit._x AND ParamInit.x = FALSE THEN
	gvl_visu.flg_btn_PosInit := FALSE;
	gvl_visu.flg_btn_PosPickUP := FALSE;
	gvl_visu.flg_btn_PosRemove := FALSE;
	gvl_visu.flg_btn_PosSample := FALSE;
	gvl_visu.flg_btn_PosPocket := FALSE;
ELSIF ParamInit._x AND ParamInit.x THEN
	flg_moveDone := FALSE;
END_IF
END_ACTION

ACTION PassPos_active:
IF PassPos._x AND PassPos.x = FALSE THEN
	trn_PassPosDone := FALSE;
	flg_moveRun := FALSE;
	fbi_CycleDelayTimer[5].IN := FALSE;
	gvl_axis.fbi_motionControler.p_Init := TRUE;
	gvl_axis.fbi_motionControler.in_flg_start := FALSE;
	gvl_axis.fbi_motionControler.in_var_direction := eP_motionDirection.XYZ;
ELSIF PassPos._x AND PassPos.x THEN
	gvl_axis.fbi_motionControler.p_Init := FALSE;
	fbi_CycleDelayTimer[5].IN := TRUE;
	IF fbi_CycleDelayTimer[5].Q THEN
		flg_moveRun := TRUE;	
	END_IF
	IF fbi_r_TRIG[5].Q THEN
		gvl_axis.fbi_motionControler.in_flg_start := TRUE;
	END_IF
	IF gvl_axis.fbi_motionControler.out_flg_Done THEN
		trn_PassPosDone := TRUE;
	END_IF
END_IF

fbi_r_TRIG[5](CLK:=flg_moveRun , Q=> );
fbi_CycleDelayTimer[5](IN:= , PT:=T#50MS , Q=> , ET=> );
END_ACTION

ACTION PosInit_active:

IF PosInit._x AND PosInit.x = FALSE THEN
	//flg reset
	trn_PosInitDone := FALSE;
	flg_moveRun := FALSE;
	fbi_CycleDelayTimer[0].IN := FALSE;
	gvl_axis.fbi_motionControler.p_Init := TRUE;
	gvl_axis.fbi_motionControler.in_flg_start := FALSE;
	//insert target postion
	gvl_axis.fbi_motionControler.in_var_targetPosX := gvl_param.var_productInfo[gvl_param.var_currentProductID].teachPos.initial.x;
	gvl_axis.fbi_motionControler.in_var_targetPosY := gvl_param.var_productInfo[gvl_param.var_currentProductID].teachPos.initial.y;
	gvl_axis.fbi_motionControler.in_var_targetPosZ := gvl_param.var_productInfo[gvl_param.var_currentProductID].teachPos.initial.z;
	gvl_axis.fbi_motionControler.in_var_direction := eP_motionDirection.XYZ;
ELSIF PosInit._x AND PosInit.x THEN
	gvl_axis.fbi_motionControler.p_Init := FALSE;
	fbi_CycleDelayTimer[0].IN := TRUE;
	IF fbi_CycleDelayTimer[0].Q THEN
		flg_moveRun := TRUE;
	END_IF
	IF fbi_r_TRIG[0].Q THEN	
		gvl_axis.fbi_motionControler.in_flg_start := TRUE;
	END_IF
	IF gvl_axis.fbi_motionControler.out_flg_Done THEN
		flg_moveRun := FALSE;
		trn_PosInitDone := TRUE;
	END_IF
	
END_IF
fbi_r_TRIG[0](CLK:=flg_moveRun , Q=> );
fbi_CycleDelayTimer[0](IN:= , PT:= T#50MS, Q=> , ET=> );
END_ACTION

ACTION PosPickUp_active:
IF PosPickUp._x AND PosPickUp.x = FALSE THEN
	//flg reset
	trn_PosPickUpDone := FALSE;
	flg_moveRun := FALSE;
	fbi_CycleDelayTimer[1].IN := FALSE;
	gvl_axis.fbi_motionControler.p_Init := TRUE;
	gvl_axis.fbi_motionControler.in_flg_start := FALSE;
	//insert target postion
	gvl_axis.fbi_motionControler.in_var_targetPosX := gvl_param.var_productInfo[gvl_param.var_currentProductID].teachPos.pickUp.x;
	gvl_axis.fbi_motionControler.in_var_targetPosY := gvl_param.var_productInfo[gvl_param.var_currentProductID].teachPos.pickUp.y;
	gvl_axis.fbi_motionControler.in_var_targetPosZ := gvl_param.var_productInfo[gvl_param.var_currentProductID].teachPos.pickUp.z;
	gvl_axis.fbi_motionControler.in_var_direction := eP_motionDirection.XYZ;
ELSIF PosPickUp._x AND PosPickUp.x THEN
	gvl_axis.fbi_motionControler.p_Init := FALSE;
	fbi_CycleDelayTimer[1].IN := TRUE;
	IF fbi_CycleDelayTimer[1].Q THEN
		flg_moveRun := TRUE;
	END_IF
	IF fbi_r_TRIG[1].Q THEN
		gvl_axis.fbi_motionControler.in_flg_start := TRUE;
	END_IF
	IF gvl_axis.fbi_motionControler.out_flg_Done THEN
		trn_PosPickUpDone := TRUE;
	END_IF
END_IF

fbi_r_TRIG[1](CLK:=flg_moveRun , Q=> );
fbi_CycleDelayTimer[1](IN:= , PT:=T#50MS , Q=> , ET=> );
END_ACTION

ACTION PosPocket_active:
IF PosPocket._x AND PosPocket.x = FALSE THEN
	//reset flag
	trn_PosPocketDone := FALSE;
	flg_moveRun := FALSE;
	fbi_CycleDelayTimer[4].IN := FALSE;
	gvl_axis.fbi_motionControler.p_Init := TRUE;
	gvl_axis.fbi_motionControler.in_flg_start := FALSE;
	gvl_axis.fbi_motionControler.in_var_direction := eP_motionDirection.XYZ;
ELSIF PosPocket._x AND PosPocket.x THEN
	gvl_axis.fbi_motionControler.p_Init := FALSE;
	fbi_CycleDelayTimer[4].IN := TRUE;
	IF fbi_CycleDelayTimer[4].Q THEN
		flg_moveRun := TRUE;	
	END_IF
	IF fbi_r_TRIG[4].Q THEN
		gvl_axis.fbi_motionControler.in_flg_start := TRUE;
	END_IF
	IF gvl_axis.fbi_motionControler.out_flg_Done THEN
		trn_PosPocketDone := TRUE;
	END_IF
END_IF

fbi_r_TRIG[4](CLK:=flg_moveRun , Q=> );
fbi_CycleDelayTimer[4](IN:= , PT:=T#50MS , Q=> , ET=> );
END_ACTION

ACTION PosRemove_active:
IF PosRemove._x AND PosRemove.x = FALSE THEN
	//flg reset
	trn_PosRemoveDone := FALSE;
	flg_moveRun := FALSE;
	fbi_CycleDelayTimer[2].IN := FALSE;
	gvl_axis.fbi_motionControler.p_Init := TRUE;
	gvl_axis.fbi_motionControler.in_flg_start := FALSE;
	//insert target postion
	gvl_axis.fbi_motionControler.in_var_targetPosX := gvl_param.var_productInfo[gvl_param.var_currentProductID].teachPos.remove.x;
	gvl_axis.fbi_motionControler.in_var_targetPosY := gvl_param.var_productInfo[gvl_param.var_currentProductID].teachPos.remove.y;
	gvl_axis.fbi_motionControler.in_var_targetPosZ := gvl_param.var_productInfo[gvl_param.var_currentProductID].teachPos.remove.z;
	gvl_axis.fbi_motionControler.in_var_direction := eP_motionDirection.XYZ;
ELSIF PosRemove._x AND PosRemove.x THEN
	gvl_axis.fbi_motionControler.p_Init := FALSE;
	fbi_CycleDelayTimer[2].IN := TRUE;
	IF fbi_CycleDelayTimer[2].Q THEN
		flg_moveRun := TRUE;
	END_IF
	IF fbi_r_TRIG[2].Q THEN
		gvl_axis.fbi_motionControler.in_flg_start := TRUE;
	END_IF
	IF gvl_axis.fbi_motionControler.out_flg_Done THEN
		trn_PosRemoveDone := TRUE;
	END_IF
END_IF

fbi_r_TRIG[2](CLK:=flg_moveRun , Q=> );
fbi_CycleDelayTimer[2](IN:= , PT:=T#50MS , Q=> , ET=> );
END_ACTION

ACTION PosSample_active:
IF PosSample._x AND PosSample.x = FALSE THEN
	//reset flag
	trn_PosSampleDone := FALSE;
	flg_moveRun := FALSE;
	fbi_CycleDelayTimer[3].IN := FALSE;
	gvl_axis.fbi_motionControler.p_Init := TRUE;
	gvl_axis.fbi_motionControler.in_flg_start := FALSE;
	//insert target postion
	gvl_axis.fbi_motionControler.in_var_targetPosX := gvl_param.var_productInfo[gvl_param.var_currentProductID].teachPos.sample[gvl_visu.var_in_sampleCavNo].x;
	gvl_axis.fbi_motionControler.in_var_targetPosX := gvl_param.var_productInfo[gvl_param.var_currentProductID].teachPos.sample[gvl_visu.var_in_sampleCavNo].y;
	gvl_axis.fbi_motionControler.in_var_targetPosX := gvl_param.var_productInfo[gvl_param.var_currentProductID].teachPos.sample[gvl_visu.var_in_sampleCavNo].z;
	gvl_axis.fbi_motionControler.in_var_direction := eP_motionDirection.XYZ;
ELSIF PosSample._x AND PosSample.x THEN
	gvl_axis.fbi_motionControler.p_Init := FALSE;
	fbi_CycleDelayTimer[3].IN := TRUE;
	IF fbi_CycleDelayTimer[3].Q THEN
		flg_moveRun := TRUE;
	END_IF
	IF fbi_r_TRIG[3].Q THEN
		gvl_axis.fbi_motionControler.in_flg_start := TRUE;
	END_IF
	IF gvl_axis.fbi_motionControler.out_flg_Done THEN
		trn_PosSampleDone := TRUE;
	END_IF
END_IF

fbi_r_TRIG[3](CLK:=flg_moveRun , Q=> );
fbi_CycleDelayTimer[3](IN:= , PT:=T#50MS , Q=> , ET=> );
END_ACTION

ACTION SetPos_active:
IF SetPos._x AND SetPos.x = FALSE THEN
	trn_SetPosDone := FALSE;
	var_process := 0;
	gvl_axis.ref_x.Position := var_targetPosX + gvl_param.var_productInfo[gvl_param.var_currentProductID].teachPos.palletize.upperLower[gvl_param.var_currentTrayPos].cav[gvl_visu.var_in_cavNo].teachingDetail.settingPOs.x;
	gvl_axis.ref_y.Position := var_targetPosY + gvl_param.var_productInfo[gvl_param.var_currentProductID].teachPos.palletize.upperLower[gvl_param.var_currentTrayPos].cav[gvl_visu.var_in_cavNo].teachingDetail.settingPOs.y;
	gvl_axis.ref_z.Position := var_targetPosZ + gvl_param.var_productInfo[gvl_param.var_currentProductID].teachPos.palletize.upperLower[gvl_param.var_currentTrayPos].cav[gvl_visu.var_in_cavNo].teachingDetail.settingPOs.z;
ELSIF SetPos._x AND SetPos.x THEN
	CASE var_process OF
		0:
			gvl_axis.ref_x.Execute := TRUE;
			gvl_axis.ref_y.Execute := TRUE;
			gvl_axis.ref_z.Execute := TRUE;
			IF gvl_axis.fbi_mc_absX.Done AND gvl_axis.fbi_mc_absY.Done AND gvl_axis.fbi_mc_absZ.Done THEN
				var_process := 1;
			END_IF
		1:
			gvl_axis.ref_x.Execute := FALSE;
			gvl_axis.ref_y.Execute := FALSE;
			gvl_axis.ref_z.Execute := FALSE;
			trn_SetPosDone := TRUE;
	END_CASE
END_IF
END_ACTION

END_FUNCTION_BLOCK

// ---- FBs/fb_coordinateCal.TcPOU
FUNCTION_BLOCK fb_coordinateCal
VAR_INPUT
	in_flg_run : BOOL;
END_VAR
VAR_OUTPUT
	out_flg_run : BOOL;	
END_VAR
VAR_IN_OUT
	var_ref_productInfo : ref_productInfo;
END_VAR
VAR_INPUT
	in_var_cavNo : INT;
	in_var_pocketNo : INT;
	in_var_calculateMode : eP_calculateMode;
END_VAR
VAR_OUTPUT

